ABB RAPID module: P43.mod

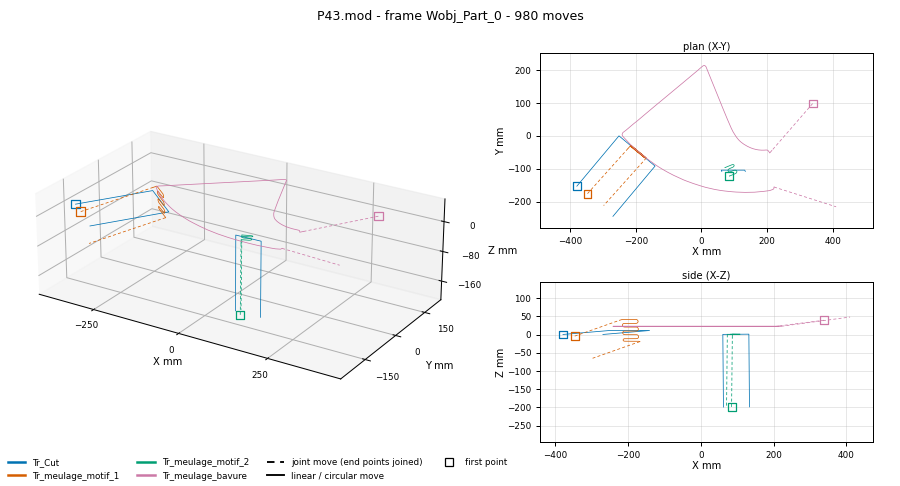
[picture p0: tool path of P43.mod in frame Wobj_Part_0, 980 of 990 moves have a stored position in this frame; points joined in program order, loops and branches not executed]
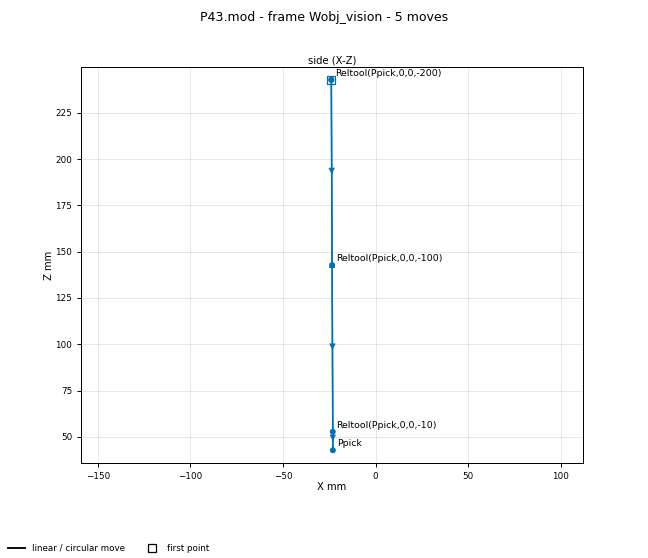
[picture p1: tool path of P43.mod in frame Wobj_vision, 5 of 990 moves have a stored position in this frame; points joined in program order, loops and branches not executed]
MODULE P43
	LOCAL CONST Speeddata vitesse_Tronconnage :=[10, 500, 0, 0];
	LOCAL CONST Robtarget Coupe_0 :=[[-192.24090625,-48.85296875,11.378640625],[0.632335428197394,0.648580331341073,0.281679878226159,0.316467859736843],[0,0,0,0],[8.999999E+09,8.999999E+09,8.999999E+09,8.999999E+09,8.999999E+09,8.999999E+09]];
	LOCAL CONST Robtarget Coupe_1 :=[[91.171640625,-104.02940625,0.997809143066406],[0.704150064324628,-0.0071021341686035,-0.709980726051425,0.00704380844178293],[0,0,0,0],[8.999999E+09,8.999999E+09,8.999999E+09,8.999999E+09,8.999999E+09,8.999999E+09]];
	LOCAL CONST Robtarget Tr_meulage_motif_1_App1 :=[[-346.886304833048,-175.614309992593,-4.01447746289841],[0.732123189175605,-0.57971865199821,0.222030212103854,-0.280400615744397],[0,0,0,0],[8.999999E+09,8.999999E+09,8.999999E+09,8.999999E+09,8.999999E+09,8.999999E+09]];
	LOCAL CONST Robtarget Tr_meulage_motif_1_App2 :=[[-223.345669929152,-37.9904471402547,39.5444929237301],[0.732123189175605,-0.57971865199821,0.222030212103854,-0.280400615744397],[0,0,0,0],[8.999999E+09,8.999999E+09,8.999999E+09,8.999999E+09,8.999999E+09,8.999999E+09]];
	LOCAL CONST Robtarget Tr_meulage_motif_1_P0 :=[[-216.84353125,-30.7470859375,41.8370703125],[0.732123189175605,-0.57971865199821,0.222030212103854,-0.280400615744397],[0,0,0,0],[8.999999E+09,8.999999E+09,8.999999E+09,8.999999E+09,8.999999E+09,8.999999E+09]];
	LOCAL CONST Robtarget Tr_meulage_motif_1_P1 :=[[-216.071953125,-31.38321875,41.837171875],[0.732123189175605,-0.57971865199821,0.222030212103854,-0.280400615744397],[0,0,0,0],[8.999999E+09,8.999999E+09,8.999999E+09,8.999999E+09,8.999999E+09,8.999999E+09]];
	LOCAL CONST Robtarget Tr_meulage_motif_1_P2 :=[[-215.300375,-32.0193515625,41.83726953125],[0.732123189175605,-0.57971865199821,0.222030212103854,-0.280400615744397],[0,0,0,0],[8.999999E+09,8.999999E+09,8.999999E+09,8.999999E+09,8.999999E+09,8.999999E+09]];
	LOCAL CONST Robtarget Tr_meulage_motif_1_P3 :=[[-214.52878125,-32.655486328125,41.8373671875],[0.732123189175605,-0.57971865199821,0.222030212103854,-0.280400615744397],[0,0,0,0],[8.999999E+09,8.999999E+09,8.999999E+09,8.999999E+09,8.999999E+09,8.999999E+09]];
	LOCAL CONST Robtarget Tr_meulage_motif_1_P4 :=[[-213.757203125,-33.2916171875,41.83746484375],[0.732123189175605,-0.57971865199821,0.222030212103854,-0.280400615744397],[0,0,0,0],[8.999999E+09,8.999999E+09,8.999999E+09,8.999999E+09,8.999999E+09,8.999999E+09]];
	LOCAL CONST Robtarget Tr_meulage_motif_1_P5 :=[[-212.985625,-33.92775390625,41.8375625],[0.732123189175605,-0.57971865199821,0.222030212103854,-0.280400615744397],[0,0,0,0],[8.999999E+09,8.999999E+09,8.999999E+09,8.999999E+09,8.999999E+09,8.999999E+09]];
	LOCAL CONST Robtarget Tr_meulage_motif_1_P6 :=[[-212.214046875,-34.56388671875,41.8376640625],[0.732123189175605,-0.57971865199821,0.222030212103854,-0.280400615744397],[0,0,0,0],[8.999999E+09,8.999999E+09,8.999999E+09,8.999999E+09,8.999999E+09,8.999999E+09]];
	LOCAL CONST Robtarget Tr_meulage_motif_1_P7 :=[[-211.44246875,-35.20001953125,41.83776171875],[0.732123189175605,-0.57971865199821,0.222030212103854,-0.280400615744397],[0,0,0,0],[8.999999E+09,8.999999E+09,8.999999E+09,8.999999E+09,8.999999E+09,8.999999E+09]];
	LOCAL CONST Robtarget Tr_meulage_motif_1_P8 :=[[-210.670890625,-35.83615234375,41.837859375],[0.732123189175605,-0.57971865199821,0.222030212103854,-0.280400615744397],[0,0,0,0],[8.999999E+09,8.999999E+09,8.999999E+09,8.999999E+09,8.999999E+09,8.999999E+09]];
	LOCAL CONST Robtarget Tr_meulage_motif_1_P9 :=[[-209.8993125,-36.47228515625,41.83795703125],[0.732123189175605,-0.57971865199821,0.222030212103854,-0.280400615744397],[0,0,0,0],[8.999999E+09,8.999999E+09,8.999999E+09,8.999999E+09,8.999999E+09,8.999999E+09]];
	LOCAL CONST Robtarget Tr_meulage_motif_1_P10 :=[[-209.127734375,-37.10841796875,41.8380546875],[0.732123189175605,-0.57971865199821,0.222030212103854,-0.280400615744397],[0,0,0,0],[8.999999E+09,8.999999E+09,8.999999E+09,8.999999E+09,8.999999E+09,8.999999E+09]];
	LOCAL CONST Robtarget Tr_meulage_motif_1_P11 :=[[-208.35615625,-37.74455078125,41.83815625],[0.732123189175605,-0.57971865199821,0.222030212103854,-0.280400615744397],[0,0,0,0],[8.999999E+09,8.999999E+09,8.999999E+09,8.999999E+09,8.999999E+09,8.999999E+09]];
	LOCAL CONST Robtarget Tr_meulage_motif_1_P12 :=[[-207.584578125,-38.38068359375,41.83825390625],[0.732123189175605,-0.57971865199821,0.222030212103854,-0.280400615744397],[0,0,0,0],[8.999999E+09,8.999999E+09,8.999999E+09,8.999999E+09,8.999999E+09,8.999999E+09]];
	LOCAL CONST Robtarget Tr_meulage_motif_1_P13 :=[[-206.813,-39.01681640625,41.8383515625],[0.732123189175605,-0.57971865199821,0.222030212103854,-0.280400615744397],[0,0,0,0],[8.999999E+09,8.999999E+09,8.999999E+09,8.999999E+09,8.999999E+09,8.999999E+09]];
	LOCAL CONST Robtarget Tr_meulage_motif_1_P14 :=[[-206.041421875,-39.65294921875,41.83844921875],[0.732123189175605,-0.57971865199821,0.222030212103854,-0.280400615744397],[0,0,0,0],[8.999999E+09,8.999999E+09,8.999999E+09,8.999999E+09,8.999999E+09,8.999999E+09]];
	LOCAL CONST Robtarget Tr_meulage_motif_1_P15 :=[[-205.26984375,-40.2890859375,41.83855078125],[0.732123189175605,-0.57971865199821,0.222030212103854,-0.280400615744397],[0,0,0,0],[8.999999E+09,8.999999E+09,8.999999E+09,8.999999E+09,8.999999E+09,8.999999E+09]];
	LOCAL CONST Robtarget Tr_meulage_motif_1_P16 :=[[-204.498265625,-40.92521875,41.8386484375],[0.732123189175605,-0.57971865199821,0.222030212103854,-0.280400615744397],[0,0,0,0],[8.999999E+09,8.999999E+09,8.999999E+09,8.999999E+09,8.999999E+09,8.999999E+09]];
	LOCAL CONST Robtarget Tr_meulage_motif_1_P17 :=[[-203.726671875,-41.5613515625,41.83874609375],[0.732123189175605,-0.57971865199821,0.222030212103854,-0.280400615744397],[0,0,0,0],[8.999999E+09,8.999999E+09,8.999999E+09,8.999999E+09,8.999999E+09,8.999999E+09]];
	LOCAL CONST Robtarget Tr_meulage_motif_1_P18 :=[[-202.95509375,-42.197484375,41.83884375],[0.732123189175605,-0.57971865199821,0.222030212103854,-0.280400615744397],[0,0,0,0],[8.999999E+09,8.999999E+09,8.999999E+09,8.999999E+09,8.999999E+09,8.999999E+09]];
	LOCAL CONST Robtarget Tr_meulage_motif_1_P19 :=[[-202.183515625,-42.8336171875,41.83894140625],[0.732123189175605,-0.57971865199821,0.222030212103854,-0.280400615744397],[0,0,0,0],[8.999999E+09,8.999999E+09,8.999999E+09,8.999999E+09,8.999999E+09,8.999999E+09]];
	LOCAL CONST Robtarget Tr_meulage_motif_1_P20 :=[[-201.4119375,-43.46975,41.83904296875],[0.732123189175605,-0.57971865199821,0.222030212103854,-0.280400615744397],[0,0,0,0],[8.999999E+09,8.999999E+09,8.999999E+09,8.999999E+09,8.999999E+09,8.999999E+09]];
	LOCAL CONST Robtarget Tr_meulage_motif_1_P21 :=[[-200.640359375,-44.1058828125,41.839140625],[0.732123189175605,-0.57971865199821,0.222030212103854,-0.280400615744397],[0,0,0,0],[8.999999E+09,8.999999E+09,8.999999E+09,8.999999E+09,8.999999E+09,8.999999E+09]];
	LOCAL CONST Robtarget Tr_meulage_motif_1_P22 :=[[-199.86878125,-44.742015625,41.83923828125],[0.732123189175605,-0.57971865199821,0.222030212103854,-0.280400615744397],[0,0,0,0],[8.999999E+09,8.999999E+09,8.999999E+09,8.999999E+09,8.999999E+09,8.999999E+09]];
	LOCAL CONST Robtarget Tr_meulage_motif_1_P23 :=[[-199.097203125,-45.3781484375,41.8393359375],[0.732123189175605,-0.57971865199821,0.222030212103854,-0.280400615744397],[0,0,0,0],[8.999999E+09,8.999999E+09,8.999999E+09,8.999999E+09,8.999999E+09,8.999999E+09]];
	LOCAL CONST Robtarget Tr_meulage_motif_1_P24 :=[[-198.325625,-46.01428515625,41.83943359375],[0.732123189175605,-0.57971865199821,0.222030212103854,-0.280400615744397],[0,0,0,0],[8.999999E+09,8.999999E+09,8.999999E+09,8.999999E+09,8.999999E+09,8.999999E+09]];
	LOCAL CONST Robtarget Tr_meulage_motif_1_P25 :=[[-197.554046875,-46.65041796875,41.83953515625],[0.732123189175605,-0.57971865199821,0.222030212103854,-0.280400615744397],[0,0,0,0],[8.999999E+09,8.999999E+09,8.999999E+09,8.999999E+09,8.999999E+09,8.999999E+09]];
	LOCAL CONST Robtarget Tr_meulage_motif_1_P26 :=[[-196.78246875,-47.28655078125,41.8396328125],[0.732123189175605,-0.57971865199821,0.222030212103854,-0.280400615744397],[0,0,0,0],[8.999999E+09,8.999999E+09,8.999999E+09,8.999999E+09,8.999999E+09,8.999999E+09]];
	LOCAL CONST Robtarget Tr_meulage_motif_1_P27 :=[[-196.010890625,-47.92268359375,41.83973046875],[0.732123189175605,-0.57971865199821,0.222030212103854,-0.280400615744397],[0,0,0,0],[8.999999E+09,8.999999E+09,8.999999E+09,8.999999E+09,8.999999E+09,8.999999E+09]];
	LOCAL CONST Robtarget Tr_meulage_motif_1_P28 :=[[-195.2393125,-48.55881640625,41.839828125],[0.732123189175605,-0.57971865199821,0.222030212103854,-0.280400615744397],[0,0,0,0],[8.999999E+09,8.999999E+09,8.999999E+09,8.999999E+09,8.999999E+09,8.999999E+09]];
	LOCAL CONST Robtarget Tr_meulage_motif_1_P29 :=[[-194.467734375,-49.19494921875,41.83992578125],[0.732123189175605,-0.57971865199821,0.222030212103854,-0.280400615744397],[0,0,0,0],[8.999999E+09,8.999999E+09,8.999999E+09,8.999999E+09,8.999999E+09,8.999999E+09]];
	LOCAL CONST Robtarget Tr_meulage_motif_1_P30 :=[[-193.69615625,-49.83108203125,41.84002734375],[0.732123189175605,-0.57971865199821,0.222030212103854,-0.280400615744397],[0,0,0,0],[8.999999E+09,8.999999E+09,8.999999E+09,8.999999E+09,8.999999E+09,8.999999E+09]];
	LOCAL CONST Robtarget Tr_meulage_motif_1_P31 :=[[-192.9245625,-50.46721484375,41.840125],[0.732123189175605,-0.57971865199821,0.222030212103854,-0.280400615744397],[0,0,0,0],[8.999999E+09,8.999999E+09,8.999999E+09,8.999999E+09,8.999999E+09,8.999999E+09]];
	LOCAL CONST Robtarget Tr_meulage_motif_1_P32 :=[[-192.152984375,-51.10334765625,41.84022265625],[0.732123189175605,-0.57971865199821,0.222030212103854,-0.280400615744397],[0,0,0,0],[8.999999E+09,8.999999E+09,8.999999E+09,8.999999E+09,8.999999E+09,8.999999E+09]];
	LOCAL CONST Robtarget Tr_meulage_motif_1_P33 :=[[-191.38140625,-51.73948046875,41.8403203125],[0.732123189175605,-0.57971865199821,0.222030212103854,-0.280400615744397],[0,0,0,0],[8.999999E+09,8.999999E+09,8.999999E+09,8.999999E+09,8.999999E+09,8.999999E+09]];
	LOCAL CONST Robtarget Tr_meulage_motif_1_P34 :=[[-190.609828125,-52.3756171875,41.840421875],[0.732123189175605,-0.57971865199821,0.222030212103854,-0.280400615744397],[0,0,0,0],[8.999999E+09,8.999999E+09,8.999999E+09,8.999999E+09,8.999999E+09,8.999999E+09]];
	LOCAL CONST Robtarget Tr_meulage_motif_1_P35 :=[[-189.83825,-53.01175,41.84051953125],[0.732123189175605,-0.57971865199821,0.222030212103854,-0.280400615744397],[0,0,0,0],[8.999999E+09,8.999999E+09,8.999999E+09,8.999999E+09,8.999999E+09,8.999999E+09]];
	LOCAL CONST Robtarget Tr_meulage_motif_1_P36 :=[[-189.066671875,-53.6478828125,41.8406171875],[0.732123189175605,-0.57971865199821,0.222030212103854,-0.280400615744397],[0,0,0,0],[8.999999E+09,8.999999E+09,8.999999E+09,8.999999E+09,8.999999E+09,8.999999E+09]];
	LOCAL CONST Robtarget Tr_meulage_motif_1_P37 :=[[-188.29509375,-54.284015625,41.84071484375],[0.732123189175605,-0.57971865199821,0.222030212103854,-0.280400615744397],[0,0,0,0],[8.999999E+09,8.999999E+09,8.999999E+09,8.999999E+09,8.999999E+09,8.999999E+09]];
	LOCAL CONST Robtarget Tr_meulage_motif_1_P38 :=[[-187.523515625,-54.9201484375,41.8408125],[0.732123189175605,-0.57971865199821,0.222030212103854,-0.280400615744397],[0,0,0,0],[8.999999E+09,8.999999E+09,8.999999E+09,8.999999E+09,8.999999E+09,8.999999E+09]];
	LOCAL CONST Robtarget Tr_meulage_motif_1_P39 :=[[-186.7519375,-55.55628125,41.8409140625],[0.732123189175605,-0.57971865199821,0.222030212103854,-0.280400615744397],[0,0,0,0],[8.999999E+09,8.999999E+09,8.999999E+09,8.999999E+09,8.999999E+09,8.999999E+09]];
	LOCAL CONST Robtarget Tr_meulage_motif_1_P40 :=[[-185.980359375,-56.1924140625,41.84101171875],[0.732123189175605,-0.57971865199821,0.222030212103854,-0.280400615744397],[0,0,0,0],[8.999999E+09,8.999999E+09,8.999999E+09,8.999999E+09,8.999999E+09,8.999999E+09]];
	LOCAL CONST Robtarget Tr_meulage_motif_1_P41 :=[[-185.20878125,-56.828546875,41.841109375],[0.732123189175605,-0.57971865199821,0.222030212103854,-0.280400615744397],[0,0,0,0],[8.999999E+09,8.999999E+09,8.999999E+09,8.999999E+09,8.999999E+09,8.999999E+09]];
	LOCAL CONST Robtarget Tr_meulage_motif_1_P42 :=[[-184.437203125,-57.4646796875,41.84120703125],[0.732123189175605,-0.57971865199821,0.222030212103854,-0.280400615744397],[0,0,0,0],[8.999999E+09,8.999999E+09,8.999999E+09,8.999999E+09,8.999999E+09,8.999999E+09]];
	LOCAL CONST Robtarget Tr_meulage_motif_1_P43 :=[[-183.665625,-58.10081640625,41.8413046875],[0.732123189175605,-0.57971865199821,0.222030212103854,-0.280400615744397],[0,0,0,0],[8.999999E+09,8.999999E+09,8.999999E+09,8.999999E+09,8.999999E+09,8.999999E+09]];
	LOCAL CONST Robtarget Tr_meulage_motif_1_P44 :=[[-182.894046875,-58.73694921875,41.84140625],[0.732123189175605,-0.57971865199821,0.222030212103854,-0.280400615744397],[0,0,0,0],[8.999999E+09,8.999999E+09,8.999999E+09,8.999999E+09,8.999999E+09,8.999999E+09]];
	LOCAL CONST Robtarget Tr_meulage_motif_1_P45 :=[[-182.122453125,-59.37308203125,41.84150390625],[0.732123189175605,-0.57971865199821,0.222030212103854,-0.280400615744397],[0,0,0,0],[8.999999E+09,8.999999E+09,8.999999E+09,8.999999E+09,8.999999E+09,8.999999E+09]];
	LOCAL CONST Robtarget Tr_meulage_motif_1_P46 :=[[-181.350875,-60.00921484375,41.8416015625],[0.732123189175605,-0.57971865199821,0.222030212103854,-0.280400615744397],[0,0,0,0],[8.999999E+09,8.999999E+09,8.999999E+09,8.999999E+09,8.999999E+09,8.999999E+09]];
	LOCAL CONST Robtarget Tr_meulage_motif_1_P47 :=[[-180.579296875,-60.64534765625,41.84169921875],[0.732123189175605,-0.57971865199821,0.222030212103854,-0.280400615744397],[0,0,0,0],[8.999999E+09,8.999999E+09,8.999999E+09,8.999999E+09,8.999999E+09,8.999999E+09]];
	LOCAL CONST Robtarget Tr_meulage_motif_1_P48 :=[[-179.80771875,-61.28148046875,41.841796875],[0.732123189175605,-0.57971865199821,0.222030212103854,-0.280400615744397],[0,0,0,0],[8.999999E+09,8.999999E+09,8.999999E+09,8.999999E+09,8.999999E+09,8.999999E+09]];
	LOCAL CONST Robtarget Tr_meulage_motif_1_P49 :=[[-179.036140625,-61.91761328125,41.8418984375],[0.732123189175605,-0.57971865199821,0.222030212103854,-0.280400615744397],[0,0,0,0],[8.999999E+09,8.999999E+09,8.999999E+09,8.999999E+09,8.999999E+09,8.999999E+09]];
	LOCAL CONST Robtarget Tr_meulage_motif_1_P50 :=[[-178.2645625,-62.55374609375,41.84199609375],[0.732123189175605,-0.57971865199821,0.222030212103854,-0.280400615744397],[0,0,0,0],[8.999999E+09,8.999999E+09,8.999999E+09,8.999999E+09,8.999999E+09,8.999999E+09]];
	LOCAL CONST Robtarget Tr_meulage_motif_1_P51 :=[[-177.49484375,-63.18045703125,41.73166796875],[0.732123189175605,-0.57971865199821,0.222030212103854,-0.280400615744397],[0,0,0,0],[8.999999E+09,8.999999E+09,8.999999E+09,8.999999E+09,8.999999E+09,8.999999E+09]];
	LOCAL CONST Robtarget Tr_meulage_motif_1_P52 :=[[-176.757125,-63.77359375,41.52089453125],[0.732123189175605,-0.57971865199821,0.222030212103854,-0.280400615744397],[0,0,0,0],[8.999999E+09,8.999999E+09,8.999999E+09,8.999999E+09,8.999999E+09,8.999999E+09]];
	LOCAL CONST Robtarget Tr_meulage_motif_1_P53 :=[[-176.089640625,-64.3045,41.249546875],[0.732123189175605,-0.57971865199821,0.222030212103854,-0.280400615744397],[0,0,0,0],[8.999999E+09,8.999999E+09,8.999999E+09,8.999999E+09,8.999999E+09,8.999999E+09]];
	LOCAL CONST Robtarget Tr_meulage_motif_1_P54 :=[[-175.5013125,-64.7698515625,40.9741015625],[0.732123189175605,-0.57971865199821,0.222030212103854,-0.280400615744397],[0,0,0,0],[8.999999E+09,8.999999E+09,8.999999E+09,8.999999E+09,8.999999E+09,8.999999E+09]];
	LOCAL CONST Robtarget Tr_meulage_motif_1_P55 :=[[-174.630125,-65.444125,40.35901953125],[0.732123189175605,-0.57971865199821,0.222030212103854,-0.280400615744397],[0,0,0,0],[8.999999E+09,8.999999E+09,8.999999E+09,8.999999E+09,8.999999E+09,8.999999E+09]];
	LOCAL CONST Robtarget Tr_meulage_motif_1_P56 :=[[-173.810359375,-66.0594765625,39.51275390625],[0.732123189175605,-0.57971865199821,0.222030212103854,-0.280400615744397],[0,0,0,0],[8.999999E+09,8.999999E+09,8.999999E+09,8.999999E+09,8.999999E+09,8.999999E+09]];
	LOCAL CONST Robtarget Tr_meulage_motif_1_P57 :=[[-173.120359375,-66.5552421875,38.490515625],[0.732123189175605,-0.57971865199821,0.222030212103854,-0.280400615744397],[0,0,0,0],[8.999999E+09,8.999999E+09,8.999999E+09,8.999999E+09,8.999999E+09,8.999999E+09]];
	LOCAL CONST Robtarget Tr_meulage_motif_1_P58 :=[[-172.704515625,-66.8184140625,37.3760703125],[0.732123189175605,-0.57971865199821,0.222030212103854,-0.280400615744397],[0,0,0,0],[8.999999E+09,8.999999E+09,8.999999E+09,8.999999E+09,8.999999E+09,8.999999E+09]];
	LOCAL CONST Robtarget Tr_meulage_motif_1_P59 :=[[-172.659203125,-66.80609375,36.68116015625],[0.732123189175605,-0.57971865199821,0.222030212103854,-0.280400615744397],[0,0,0,0],[8.999999E+09,8.999999E+09,8.999999E+09,8.999999E+09,8.999999E+09,8.999999E+09]];
	LOCAL CONST Robtarget Tr_meulage_motif_1_P60 :=[[-172.635984375,-66.77803125,36.0209140625],[0.732123189175605,-0.57971865199821,0.222030212103854,-0.280400615744397],[0,0,0,0],[8.999999E+09,8.999999E+09,8.999999E+09,8.999999E+09,8.999999E+09,8.999999E+09]];
	LOCAL CONST Robtarget Tr_meulage_motif_1_P61 :=[[-172.655109375,-66.7150625,35.3608203125],[0.732123189175605,-0.57971865199821,0.222030212103854,-0.280400615744397],[0,0,0,0],[8.999999E+09,8.999999E+09,8.999999E+09,8.999999E+09,8.999999E+09,8.999999E+09]];
	LOCAL CONST Robtarget Tr_meulage_motif_1_P62 :=[[-173.000828125,-66.351375,34.26069140625],[0.732123189175605,-0.57971865199821,0.222030212103854,-0.280400615744397],[0,0,0,0],[8.999999E+09,8.999999E+09,8.999999E+09,8.999999E+09,8.999999E+09,8.999999E+09]];
	LOCAL CONST Robtarget Tr_meulage_motif_1_P63 :=[[-173.6264375,-65.763734375,33.25551171875],[0.732123189175605,-0.57971865199821,0.222030212103854,-0.280400615744397],[0,0,0,0],[8.999999E+09,8.999999E+09,8.999999E+09,8.999999E+09,8.999999E+09,8.999999E+09]];
	LOCAL CONST Robtarget Tr_meulage_motif_1_P64 :=[[-174.38696875,-65.07753125,32.427794921875],[0.732123189175605,-0.57971865199821,0.222030212103854,-0.280400615744397],[0,0,0,0],[8.999999E+09,8.999999E+09,8.999999E+09,8.999999E+09,8.999999E+09,8.999999E+09]];
	LOCAL CONST Robtarget Tr_meulage_motif_1_P65 :=[[-174.90321875,-64.62365625,32.032578125],[0.732123189175605,-0.57971865199821,0.222030212103854,-0.280400615744397],[0,0,0,0],[8.999999E+09,8.999999E+09,8.999999E+09,8.999999E+09,8.999999E+09,8.999999E+09]];
	LOCAL CONST Robtarget Tr_meulage_motif_1_P66 :=[[-175.77971875,-63.86622265625,31.545671875],[0.732123189175605,-0.57971865199821,0.222030212103854,-0.280400615744397],[0,0,0,0],[8.999999E+09,8.999999E+09,8.999999E+09,8.999999E+09,8.999999E+09,8.999999E+09]];
	LOCAL CONST Robtarget Tr_meulage_motif_1_P67 :=[[-176.422453125,-63.31746484375,31.281896484375],[0.732123189175605,-0.57971865199821,0.222030212103854,-0.280400615744397],[0,0,0,0],[8.999999E+09,8.999999E+09,8.999999E+09,8.999999E+09,8.999999E+09,8.999999E+09]];
	LOCAL CONST Robtarget Tr_meulage_motif_1_P68 :=[[-177.134375,-62.71591015625,31.077646484375],[0.732123189175605,-0.57971865199821,0.222030212103854,-0.280400615744397],[0,0,0,0],[8.999999E+09,8.999999E+09,8.999999E+09,8.999999E+09,8.999999E+09,8.999999E+09]];
	LOCAL CONST Robtarget Tr_meulage_motif_1_P69 :=[[-177.887921875,-62.0868984375,30.96912109375],[0.732123189175605,-0.57971865199821,0.222030212103854,-0.280400615744397],[0,0,0,0],[8.999999E+09,8.999999E+09,8.999999E+09,8.999999E+09,8.999999E+09,8.999999E+09]];
	LOCAL CONST Robtarget Tr_meulage_motif_1_P70 :=[[-178.649875,-61.45080078125,30.85859765625],[0.732123189175605,-0.57971865199821,0.222030212103854,-0.280400615744397],[0,0,0,0],[8.999999E+09,8.999999E+09,8.999999E+09,8.999999E+09,8.999999E+09,8.999999E+09]];
	LOCAL CONST Robtarget Tr_meulage_motif_1_P71 :=[[-179.421453125,-60.81466796875,30.858498046875],[0.732123189175605,-0.57971865199821,0.222030212103854,-0.280400615744397],[0,0,0,0],[8.999999E+09,8.999999E+09,8.999999E+09,8.999999E+09,8.999999E+09,8.999999E+09]];
	LOCAL CONST Robtarget Tr_meulage_motif_1_P72 :=[[-180.19303125,-60.17853515625,30.858400390625],[0.732123189175605,-0.57971865199821,0.222030212103854,-0.280400615744397],[0,0,0,0],[8.999999E+09,8.999999E+09,8.999999E+09,8.999999E+09,8.999999E+09,8.999999E+09]];
	LOCAL CONST Robtarget Tr_meulage_motif_1_P73 :=[[-180.964609375,-59.54240234375,30.85830078125],[0.732123189175605,-0.57971865199821,0.222030212103854,-0.280400615744397],[0,0,0,0],[8.999999E+09,8.999999E+09,8.999999E+09,8.999999E+09,8.999999E+09,8.999999E+09]];
	LOCAL CONST Robtarget Tr_meulage_motif_1_P74 :=[[-181.7361875,-58.90626953125,30.858203125],[0.732123189175605,-0.57971865199821,0.222030212103854,-0.280400615744397],[0,0,0,0],[8.999999E+09,8.999999E+09,8.999999E+09,8.999999E+09,8.999999E+09,8.999999E+09]];
	LOCAL CONST Robtarget Tr_meulage_motif_1_P75 :=[[-182.507765625,-58.27013671875,30.858103515625],[0.732123189175605,-0.57971865199821,0.222030212103854,-0.280400615744397],[0,0,0,0],[8.999999E+09,8.999999E+09,8.999999E+09,8.999999E+09,8.999999E+09,8.999999E+09]];
	LOCAL CONST Robtarget Tr_meulage_motif_1_P76 :=[[-183.279359375,-57.63400390625,30.858005859375],[0.732123189175605,-0.57971865199821,0.222030212103854,-0.280400615744397],[0,0,0,0],[8.999999E+09,8.999999E+09,8.999999E+09,8.999999E+09,8.999999E+09,8.999999E+09]];
	LOCAL CONST Robtarget Tr_meulage_motif_1_P77 :=[[-184.0509375,-56.99787109375,30.857908203125],[0.732123189175605,-0.57971865199821,0.222030212103854,-0.280400615744397],[0,0,0,0],[8.999999E+09,8.999999E+09,8.999999E+09,8.999999E+09,8.999999E+09,8.999999E+09]];
	LOCAL CONST Robtarget Tr_meulage_motif_1_P78 :=[[-184.822515625,-56.36173828125,30.85780859375],[0.732123189175605,-0.57971865199821,0.222030212103854,-0.280400615744397],[0,0,0,0],[8.999999E+09,8.999999E+09,8.999999E+09,8.999999E+09,8.999999E+09,8.999999E+09]];
	LOCAL CONST Robtarget Tr_meulage_motif_1_P79 :=[[-185.59409375,-55.7256015625,30.8577109375],[0.732123189175605,-0.57971865199821,0.222030212103854,-0.280400615744397],[0,0,0,0],[8.999999E+09,8.999999E+09,8.999999E+09,8.999999E+09,8.999999E+09,8.999999E+09]];
	LOCAL CONST Robtarget Tr_meulage_motif_1_P80 :=[[-186.365671875,-55.08946875,30.857611328125],[0.732123189175605,-0.57971865199821,0.222030212103854,-0.280400615744397],[0,0,0,0],[8.999999E+09,8.999999E+09,8.999999E+09,8.999999E+09,8.999999E+09,8.999999E+09]];
	LOCAL CONST Robtarget Tr_meulage_motif_1_P81 :=[[-187.13725,-54.4533359375,30.857513671875],[0.732123189175605,-0.57971865199821,0.222030212103854,-0.280400615744397],[0,0,0,0],[8.999999E+09,8.999999E+09,8.999999E+09,8.999999E+09,8.999999E+09,8.999999E+09]];
	LOCAL CONST Robtarget Tr_meulage_motif_1_P82 :=[[-187.908828125,-53.817203125,30.857416015625],[0.732123189175605,-0.57971865199821,0.222030212103854,-0.280400615744397],[0,0,0,0],[8.999999E+09,8.999999E+09,8.999999E+09,8.999999E+09,8.999999E+09,8.999999E+09]];
	LOCAL CONST Robtarget Tr_meulage_motif_1_P83 :=[[-188.68040625,-53.1810703125,30.85731640625],[0.732123189175605,-0.57971865199821,0.222030212103854,-0.280400615744397],[0,0,0,0],[8.999999E+09,8.999999E+09,8.999999E+09,8.999999E+09,8.999999E+09,8.999999E+09]];
	LOCAL CONST Robtarget Tr_meulage_motif_1_P84 :=[[-189.451984375,-52.5449375,30.85721875],[0.732123189175605,-0.57971865199821,0.222030212103854,-0.280400615744397],[0,0,0,0],[8.999999E+09,8.999999E+09,8.999999E+09,8.999999E+09,8.999999E+09,8.999999E+09]];
	LOCAL CONST Robtarget Tr_meulage_motif_1_P85 :=[[-190.2235625,-51.9088046875,30.857119140625],[0.732123189175605,-0.57971865199821,0.222030212103854,-0.280400615744397],[0,0,0,0],[8.999999E+09,8.999999E+09,8.999999E+09,8.999999E+09,8.999999E+09,8.999999E+09]];
	LOCAL CONST Robtarget Tr_meulage_motif_1_P86 :=[[-190.995140625,-51.272671875,30.857021484375],[0.732123189175605,-0.57971865199821,0.222030212103854,-0.280400615744397],[0,0,0,0],[8.999999E+09,8.999999E+09,8.999999E+09,8.999999E+09,8.999999E+09,8.999999E+09]];
	LOCAL CONST Robtarget Tr_meulage_motif_1_P87 :=[[-191.76671875,-50.6365390625,30.856921875],[0.732123189175605,-0.57971865199821,0.222030212103854,-0.280400615744397],[0,0,0,0],[8.999999E+09,8.999999E+09,8.999999E+09,8.999999E+09,8.999999E+09,8.999999E+09]];
	LOCAL CONST Robtarget Tr_meulage_motif_1_P88 :=[[-192.538296875,-50.00040625,30.85682421875],[0.732123189175605,-0.57971865199821,0.222030212103854,-0.280400615744397],[0,0,0,0],[8.999999E+09,8.999999E+09,8.999999E+09,8.999999E+09,8.999999E+09,8.999999E+09]];
	LOCAL CONST Robtarget Tr_meulage_motif_1_P89 :=[[-193.309875,-49.36426953125,30.8567265625],[0.732123189175605,-0.57971865199821,0.222030212103854,-0.280400615744397],[0,0,0,0],[8.999999E+09,8.999999E+09,8.999999E+09,8.999999E+09,8.999999E+09,8.999999E+09]];
	LOCAL CONST Robtarget Tr_meulage_motif_1_P90 :=[[-194.08146875,-48.72813671875,30.856626953125],[0.732123189175605,-0.57971865199821,0.222030212103854,-0.280400615744397],[0,0,0,0],[8.999999E+09,8.999999E+09,8.999999E+09,8.999999E+09,8.999999E+09,8.999999E+09]];
	LOCAL CONST Robtarget Tr_meulage_motif_1_P91 :=[[-194.853046875,-48.09200390625,30.856529296875],[0.732123189175605,-0.57971865199821,0.222030212103854,-0.280400615744397],[0,0,0,0],[8.999999E+09,8.999999E+09,8.999999E+09,8.999999E+09,8.999999E+09,8.999999E+09]];
	LOCAL CONST Robtarget Tr_meulage_motif_1_P92 :=[[-195.624625,-47.45587109375,30.8564296875],[0.732123189175605,-0.57971865199821,0.222030212103854,-0.280400615744397],[0,0,0,0],[8.999999E+09,8.999999E+09,8.999999E+09,8.999999E+09,8.999999E+09,8.999999E+09]];
	LOCAL CONST Robtarget Tr_meulage_motif_1_P93 :=[[-196.396203125,-46.81973828125,30.85633203125],[0.732123189175605,-0.57971865199821,0.222030212103854,-0.280400615744397],[0,0,0,0],[8.999999E+09,8.999999E+09,8.999999E+09,8.999999E+09,8.999999E+09,8.999999E+09]];
	LOCAL CONST Robtarget Tr_meulage_motif_1_P94 :=[[-197.16778125,-46.18360546875,30.856234375],[0.732123189175605,-0.57971865199821,0.222030212103854,-0.280400615744397],[0,0,0,0],[8.999999E+09,8.999999E+09,8.999999E+09,8.999999E+09,8.999999E+09,8.999999E+09]];
	LOCAL CONST Robtarget Tr_meulage_motif_1_P95 :=[[-197.939359375,-45.54747265625,30.856134765625],[0.732123189175605,-0.57971865199821,0.222030212103854,-0.280400615744397],[0,0,0,0],[8.999999E+09,8.999999E+09,8.999999E+09,8.999999E+09,8.999999E+09,8.999999E+09]];
	LOCAL CONST Robtarget Tr_meulage_motif_1_P96 :=[[-198.7109375,-44.91133984375,30.856037109375],[0.732123189175605,-0.57971865199821,0.222030212103854,-0.280400615744397],[0,0,0,0],[8.999999E+09,8.999999E+09,8.999999E+09,8.999999E+09,8.999999E+09,8.999999E+09]];
	LOCAL CONST Robtarget Tr_meulage_motif_1_P97 :=[[-199.482515625,-44.27520703125,30.8559375],[0.732123189175605,-0.57971865199821,0.222030212103854,-0.280400615744397],[0,0,0,0],[8.999999E+09,8.999999E+09,8.999999E+09,8.999999E+09,8.999999E+09,8.999999E+09]];
	LOCAL CONST Robtarget Tr_meulage_motif_1_P98 :=[[-200.25409375,-43.6390703125,30.85583984375],[0.732123189175605,-0.57971865199821,0.222030212103854,-0.280400615744397],[0,0,0,0],[8.999999E+09,8.999999E+09,8.999999E+09,8.999999E+09,8.999999E+09,8.999999E+09]];
	LOCAL CONST Robtarget Tr_meulage_motif_1_P99 :=[[-201.025671875,-43.0029375,30.855740234375],[0.732123189175605,-0.57971865199821,0.222030212103854,-0.280400615744397],[0,0,0,0],[8.999999E+09,8.999999E+09,8.999999E+09,8.999999E+09,8.999999E+09,8.999999E+09]];
	LOCAL CONST Robtarget Tr_meulage_motif_1_P100 :=[[-201.79725,-42.3668046875,30.855642578125],[0.732123189175605,-0.57971865199821,0.222030212103854,-0.280400615744397],[0,0,0,0],[8.999999E+09,8.999999E+09,8.999999E+09,8.999999E+09,8.999999E+09,8.999999E+09]];
	LOCAL CONST Robtarget Tr_meulage_motif_1_P101 :=[[-202.568828125,-41.730671875,30.855544921875],[0.732123189175605,-0.57971865199821,0.222030212103854,-0.280400615744397],[0,0,0,0],[8.999999E+09,8.999999E+09,8.999999E+09,8.999999E+09,8.999999E+09,8.999999E+09]];
	LOCAL CONST Robtarget Tr_meulage_motif_1_P102 :=[[-203.34040625,-41.0945390625,30.8554453125],[0.732123189175605,-0.57971865199821,0.222030212103854,-0.280400615744397],[0,0,0,0],[8.999999E+09,8.999999E+09,8.999999E+09,8.999999E+09,8.999999E+09,8.999999E+09]];
	LOCAL CONST Robtarget Tr_meulage_motif_1_P103 :=[[-204.111984375,-40.45840625,30.85534765625],[0.732123189175605,-0.57971865199821,0.222030212103854,-0.280400615744397],[0,0,0,0],[8.999999E+09,8.999999E+09,8.999999E+09,8.999999E+09,8.999999E+09,8.999999E+09]];
	LOCAL CONST Robtarget Tr_meulage_motif_1_P104 :=[[-204.883578125,-39.8222734375,30.855248046875],[0.732123189175605,-0.57971865199821,0.222030212103854,-0.280400615744397],[0,0,0,0],[8.999999E+09,8.999999E+09,8.999999E+09,8.999999E+09,8.999999E+09,8.999999E+09]];
	LOCAL CONST Robtarget Tr_meulage_motif_1_P105 :=[[-205.65515625,-39.186140625,30.855150390625],[0.732123189175605,-0.57971865199821,0.222030212103854,-0.280400615744397],[0,0,0,0],[8.999999E+09,8.999999E+09,8.999999E+09,8.999999E+09,8.999999E+09,8.999999E+09]];
	LOCAL CONST Robtarget Tr_meulage_motif_1_P106 :=[[-206.426734375,-38.5500078125,30.85505078125],[0.732123189175605,-0.57971865199821,0.222030212103854,-0.280400615744397],[0,0,0,0],[8.999999E+09,8.999999E+09,8.999999E+09,8.999999E+09,8.999999E+09,8.999999E+09]];
	LOCAL CONST Robtarget Tr_meulage_motif_1_P107 :=[[-207.1983125,-37.913875,30.854953125],[0.732123189175605,-0.57971865199821,0.222030212103854,-0.280400615744397],[0,0,0,0],[8.999999E+09,8.999999E+09,8.999999E+09,8.999999E+09,8.999999E+09,8.999999E+09]];
	LOCAL CONST Robtarget Tr_meulage_motif_1_P108 :=[[-207.969890625,-37.27773828125,30.85485546875],[0.732123189175605,-0.57971865199821,0.222030212103854,-0.280400615744397],[0,0,0,0],[8.999999E+09,8.999999E+09,8.999999E+09,8.999999E+09,8.999999E+09,8.999999E+09]];
	LOCAL CONST Robtarget Tr_meulage_motif_1_P109 :=[[-208.74146875,-36.64160546875,30.854755859375],[0.732123189175605,-0.57971865199821,0.222030212103854,-0.280400615744397],[0,0,0,0],[8.999999E+09,8.999999E+09,8.999999E+09,8.999999E+09,8.999999E+09,8.999999E+09]];
	LOCAL CONST Robtarget Tr_meulage_motif_1_P110 :=[[-209.513046875,-36.00547265625,30.854658203125],[0.732123189175605,-0.57971865199821,0.222030212103854,-0.280400615744397],[0,0,0,0],[8.999999E+09,8.999999E+09,8.999999E+09,8.999999E+09,8.999999E+09,8.999999E+09]];
	LOCAL CONST Robtarget Tr_meulage_motif_1_P111 :=[[-210.284625,-35.36933984375,30.85455859375],[0.732123189175605,-0.57971865199821,0.222030212103854,-0.280400615744397],[0,0,0,0],[8.999999E+09,8.999999E+09,8.999999E+09,8.999999E+09,8.999999E+09,8.999999E+09]];
	LOCAL CONST Robtarget Tr_meulage_motif_1_P112 :=[[-211.056203125,-34.73320703125,30.8544609375],[0.732123189175605,-0.57971865199821,0.222030212103854,-0.280400615744397],[0,0,0,0],[8.999999E+09,8.999999E+09,8.999999E+09,8.999999E+09,8.999999E+09,8.999999E+09]];
	LOCAL CONST Robtarget Tr_meulage_motif_1_P113 :=[[-211.81815625,-34.09711328125,30.7439375],[0.732123189175605,-0.57971865199821,0.222030212103854,-0.280400615744397],[0,0,0,0],[8.999999E+09,8.999999E+09,8.999999E+09,8.999999E+09,8.999999E+09,8.999999E+09]];
	LOCAL CONST Robtarget Tr_meulage_motif_1_P114 :=[[-212.541046875,-33.48605078125,30.5329765625],[0.732123189175605,-0.57971865199821,0.222030212103854,-0.280400615744397],[0,0,0,0],[8.999999E+09,8.999999E+09,8.999999E+09,8.999999E+09,8.999999E+09,8.999999E+09]];
	LOCAL CONST Robtarget Tr_meulage_motif_1_P115 :=[[-213.1894375,-32.9320703125,30.261462890625],[0.732123189175605,-0.57971865199821,0.222030212103854,-0.280400615744397],[0,0,0,0],[8.999999E+09,8.999999E+09,8.999999E+09,8.999999E+09,8.999999E+09,8.999999E+09]];
	LOCAL CONST Robtarget Tr_meulage_motif_1_P116 :=[[-213.727734375,-32.4665546875,29.957697265625],[0.732123189175605,-0.57971865199821,0.222030212103854,-0.280400615744397],[0,0,0,0],[8.999999E+09,8.999999E+09,8.999999E+09,8.999999E+09,8.999999E+09,8.999999E+09]];
	LOCAL CONST Robtarget Tr_meulage_motif_1_P117 :=[[-214.502640625,-31.78037890625,29.2960703125],[0.732123189175605,-0.57971865199821,0.222030212103854,-0.280400615744397],[0,0,0,0],[8.999999E+09,8.999999E+09,8.999999E+09,8.999999E+09,8.999999E+09,8.999999E+09]];
	LOCAL CONST Robtarget Tr_meulage_motif_1_P118 :=[[-215.166890625,-31.168349609375,28.3954140625],[0.732123189175605,-0.57971865199821,0.222030212103854,-0.280400615744397],[0,0,0,0],[8.999999E+09,8.999999E+09,8.999999E+09,8.999999E+09,8.999999E+09,8.999999E+09]];
	LOCAL CONST Robtarget Tr_meulage_motif_1_P119 :=[[-215.5429375,-30.783646484375,27.35091796875],[0.732123189175605,-0.57971865199821,0.222030212103854,-0.280400615744397],[0,0,0,0],[8.999999E+09,8.999999E+09,8.999999E+09,8.999999E+09,8.999999E+09,8.999999E+09]];
	LOCAL CONST Robtarget Tr_meulage_motif_1_P120 :=[[-215.66115625,-30.63668359375,26.658732421875],[0.732123189175605,-0.57971865199821,0.222030212103854,-0.280400615744397],[0,0,0,0],[8.999999E+09,8.999999E+09,8.999999E+09,8.999999E+09,8.999999E+09,8.999999E+09]];
	LOCAL CONST Robtarget Tr_meulage_motif_1_P121 :=[[-215.683390625,-30.56339453125,25.889896484375],[0.732123189175605,-0.57971865199821,0.222030212103854,-0.280400615744397],[0,0,0,0],[8.999999E+09,8.999999E+09,8.999999E+09,8.999999E+09,8.999999E+09,8.999999E+09]];
	LOCAL CONST Robtarget Tr_meulage_motif_1_P122 :=[[-215.604703125,-30.573302734375,25.1211953125],[0.732123189175605,-0.57971865199821,0.222030212103854,-0.280400615744397],[0,0,0,0],[8.999999E+09,8.999999E+09,8.999999E+09,8.999999E+09,8.999999E+09,8.999999E+09]];
	LOCAL CONST Robtarget Tr_meulage_motif_1_P123 :=[[-215.24203125,-30.793189453125,24.014669921875],[0.732123189175605,-0.57971865199821,0.222030212103854,-0.280400615744397],[0,0,0,0],[8.999999E+09,8.999999E+09,8.999999E+09,8.999999E+09,8.999999E+09,8.999999E+09]];
	LOCAL CONST Robtarget Tr_meulage_motif_1_P124 :=[[-214.901796875,-31.031892578125,23.429912109375],[0.732123189175605,-0.57971865199821,0.222030212103854,-0.280400615744397],[0,0,0,0],[8.999999E+09,8.999999E+09,8.999999E+09,8.999999E+09,8.999999E+09,8.999999E+09]];
	LOCAL CONST Robtarget Tr_meulage_motif_1_P125 :=[[-214.18615625,-31.55857421875,22.544220703125],[0.732123189175605,-0.57971865199821,0.222030212103854,-0.280400615744397],[0,0,0,0],[8.999999E+09,8.999999E+09,8.999999E+09,8.999999E+09,8.999999E+09,8.999999E+09]];
	LOCAL CONST Robtarget Tr_meulage_motif_1_P126 :=[[-213.719703125,-31.913568359375,22.130595703125],[0.732123189175605,-0.57971865199821,0.222030212103854,-0.280400615744397],[0,0,0,0],[8.999999E+09,8.999999E+09,8.999999E+09,8.999999E+09,8.999999E+09,8.999999E+09]];
	LOCAL CONST Robtarget Tr_meulage_motif_1_P127 :=[[-212.838046875,-32.601615234375,21.5874375],[0.732123189175605,-0.57971865199821,0.222030212103854,-0.280400615744397],[0,0,0,0],[8.999999E+09,8.999999E+09,8.999999E+09,8.999999E+09,8.999999E+09,8.999999E+09]];
	LOCAL CONST Robtarget Tr_meulage_motif_1_P128 :=[[-212.19065625,-33.11426171875,21.29246875],[0.732123189175605,-0.57971865199821,0.222030212103854,-0.280400615744397],[0,0,0,0],[8.999999E+09,8.999999E+09,8.999999E+09,8.999999E+09,8.999999E+09,8.999999E+09]];
	LOCAL CONST Robtarget Tr_meulage_motif_1_P129 :=[[-211.464359375,-33.6984609375,21.088400390625],[0.732123189175605,-0.57971865199821,0.222030212103854,-0.280400615744397],[0,0,0,0],[8.999999E+09,8.999999E+09,8.999999E+09,8.999999E+09,8.999999E+09,8.999999E+09]];
	LOCAL CONST Robtarget Tr_meulage_motif_1_P130 :=[[-210.703203125,-34.3182578125,20.980068359375],[0.732123189175605,-0.57971865199821,0.222030212103854,-0.280400615744397],[0,0,0,0],[8.999999E+09,8.999999E+09,8.999999E+09,8.999999E+09,8.999999E+09,8.999999E+09]];
	LOCAL CONST Robtarget Tr_meulage_motif_1_P131 :=[[-209.93346875,-34.94496484375,20.869740234375],[0.732123189175605,-0.57971865199821,0.222030212103854,-0.280400615744397],[0,0,0,0],[8.999999E+09,8.999999E+09,8.999999E+09,8.999999E+09,8.999999E+09,8.999999E+09]];
	LOCAL CONST Robtarget Tr_meulage_motif_1_P132 :=[[-209.161890625,-35.58109765625,20.86983984375],[0.732123189175605,-0.57971865199821,0.222030212103854,-0.280400615744397],[0,0,0,0],[8.999999E+09,8.999999E+09,8.999999E+09,8.999999E+09,8.999999E+09,8.999999E+09]];
	LOCAL CONST Robtarget Tr_meulage_motif_1_P133 :=[[-208.3903125,-36.217234375,20.8699375],[0.732123189175605,-0.57971865199821,0.222030212103854,-0.280400615744397],[0,0,0,0],[8.999999E+09,8.999999E+09,8.999999E+09,8.999999E+09,8.999999E+09,8.999999E+09]];
	LOCAL CONST Robtarget Tr_meulage_motif_1_P134 :=[[-207.618734375,-36.8533671875,20.870037109375],[0.732123189175605,-0.57971865199821,0.222030212103854,-0.280400615744397],[0,0,0,0],[8.999999E+09,8.999999E+09,8.999999E+09,8.999999E+09,8.999999E+09,8.999999E+09]];
	LOCAL CONST Robtarget Tr_meulage_motif_1_P135 :=[[-206.84715625,-37.4895,20.870134765625],[0.732123189175605,-0.57971865199821,0.222030212103854,-0.280400615744397],[0,0,0,0],[8.999999E+09,8.999999E+09,8.999999E+09,8.999999E+09,8.999999E+09,8.999999E+09]];
	LOCAL CONST Robtarget Tr_meulage_motif_1_P136 :=[[-206.075578125,-38.1256328125,20.870232421875],[0.732123189175605,-0.57971865199821,0.222030212103854,-0.280400615744397],[0,0,0,0],[8.999999E+09,8.999999E+09,8.999999E+09,8.999999E+09,8.999999E+09,8.999999E+09]];
	LOCAL CONST Robtarget Tr_meulage_motif_1_P137 :=[[-205.304,-38.761765625,20.87033203125],[0.732123189175605,-0.57971865199821,0.222030212103854,-0.280400615744397],[0,0,0,0],[8.999999E+09,8.999999E+09,8.999999E+09,8.999999E+09,8.999999E+09,8.999999E+09]];
	LOCAL CONST Robtarget Tr_meulage_motif_1_P138 :=[[-204.532421875,-39.3978984375,20.8704296875],[0.732123189175605,-0.57971865199821,0.222030212103854,-0.280400615744397],[0,0,0,0],[8.999999E+09,8.999999E+09,8.999999E+09,8.999999E+09,8.999999E+09,8.999999E+09]];
	LOCAL CONST Robtarget Tr_meulage_motif_1_P139 :=[[-203.76084375,-40.03403125,20.870529296875],[0.732123189175605,-0.57971865199821,0.222030212103854,-0.280400615744397],[0,0,0,0],[8.999999E+09,8.999999E+09,8.999999E+09,8.999999E+09,8.999999E+09,8.999999E+09]];
	LOCAL CONST Robtarget Tr_meulage_motif_1_P140 :=[[-202.989265625,-40.6701640625,20.870626953125],[0.732123189175605,-0.57971865199821,0.222030212103854,-0.280400615744397],[0,0,0,0],[8.999999E+09,8.999999E+09,8.999999E+09,8.999999E+09,8.999999E+09,8.999999E+09]];
	LOCAL CONST Robtarget Tr_meulage_motif_1_P141 :=[[-202.2176875,-41.306296875,20.8707265625],[0.732123189175605,-0.57971865199821,0.222030212103854,-0.280400615744397],[0,0,0,0],[8.999999E+09,8.999999E+09,8.999999E+09,8.999999E+09,8.999999E+09,8.999999E+09]];
	LOCAL CONST Robtarget Tr_meulage_motif_1_P142 :=[[-201.44609375,-41.94243359375,20.87082421875],[0.732123189175605,-0.57971865199821,0.222030212103854,-0.280400615744397],[0,0,0,0],[8.999999E+09,8.999999E+09,8.999999E+09,8.999999E+09,8.999999E+09,8.999999E+09]];
	LOCAL CONST Robtarget Tr_meulage_motif_1_P143 :=[[-200.674515625,-42.57856640625,20.870921875],[0.732123189175605,-0.57971865199821,0.222030212103854,-0.280400615744397],[0,0,0,0],[8.999999E+09,8.999999E+09,8.999999E+09,8.999999E+09,8.999999E+09,8.999999E+09]];
	LOCAL CONST Robtarget Tr_meulage_motif_1_P144 :=[[-199.9029375,-43.21469921875,20.871021484375],[0.732123189175605,-0.57971865199821,0.222030212103854,-0.280400615744397],[0,0,0,0],[8.999999E+09,8.999999E+09,8.999999E+09,8.999999E+09,8.999999E+09,8.999999E+09]];
	LOCAL CONST Robtarget Tr_meulage_motif_1_P145 :=[[-199.131359375,-43.85083203125,20.871119140625],[0.732123189175605,-0.57971865199821,0.222030212103854,-0.280400615744397],[0,0,0,0],[8.999999E+09,8.999999E+09,8.999999E+09,8.999999E+09,8.999999E+09,8.999999E+09]];
	LOCAL CONST Robtarget Tr_meulage_motif_1_P146 :=[[-198.35978125,-44.48696484375,20.87121875],[0.732123189175605,-0.57971865199821,0.222030212103854,-0.280400615744397],[0,0,0,0],[8.999999E+09,8.999999E+09,8.999999E+09,8.999999E+09,8.999999E+09,8.999999E+09]];
	LOCAL CONST Robtarget Tr_meulage_motif_1_P147 :=[[-197.588203125,-45.12309765625,20.87131640625],[0.732123189175605,-0.57971865199821,0.222030212103854,-0.280400615744397],[0,0,0,0],[8.999999E+09,8.999999E+09,8.999999E+09,8.999999E+09,8.999999E+09,8.999999E+09]];
	LOCAL CONST Robtarget Tr_meulage_motif_1_P148 :=[[-196.816625,-45.75923046875,20.8714140625],[0.732123189175605,-0.57971865199821,0.222030212103854,-0.280400615744397],[0,0,0,0],[8.999999E+09,8.999999E+09,8.999999E+09,8.999999E+09,8.999999E+09,8.999999E+09]];
	LOCAL CONST Robtarget Tr_meulage_motif_1_P149 :=[[-196.045046875,-46.39536328125,20.871513671875],[0.732123189175605,-0.57971865199821,0.222030212103854,-0.280400615744397],[0,0,0,0],[8.999999E+09,8.999999E+09,8.999999E+09,8.999999E+09,8.999999E+09,8.999999E+09]];
	LOCAL CONST Robtarget Tr_meulage_motif_1_P150 :=[[-195.27346875,-47.03149609375,20.871611328125],[0.732123189175605,-0.57971865199821,0.222030212103854,-0.280400615744397],[0,0,0,0],[8.999999E+09,8.999999E+09,8.999999E+09,8.999999E+09,8.999999E+09,8.999999E+09]];
	LOCAL CONST Robtarget Tr_meulage_motif_1_P151 :=[[-194.501890625,-47.66762890625,20.8717109375],[0.732123189175605,-0.57971865199821,0.222030212103854,-0.280400615744397],[0,0,0,0],[8.999999E+09,8.999999E+09,8.999999E+09,8.999999E+09,8.999999E+09,8.999999E+09]];
	LOCAL CONST Robtarget Tr_meulage_motif_1_P152 :=[[-193.7303125,-48.303765625,20.87180859375],[0.732123189175605,-0.57971865199821,0.222030212103854,-0.280400615744397],[0,0,0,0],[8.999999E+09,8.999999E+09,8.999999E+09,8.999999E+09,8.999999E+09,8.999999E+09]];
	LOCAL CONST Robtarget Tr_meulage_motif_1_P153 :=[[-192.958734375,-48.9398984375,20.871908203125],[0.732123189175605,-0.57971865199821,0.222030212103854,-0.280400615744397],[0,0,0,0],[8.999999E+09,8.999999E+09,8.999999E+09,8.999999E+09,8.999999E+09,8.999999E+09]];
	LOCAL CONST Robtarget Tr_meulage_motif_1_P154 :=[[-192.18715625,-49.57603125,20.872005859375],[0.732123189175605,-0.57971865199821,0.222030212103854,-0.280400615744397],[0,0,0,0],[8.999999E+09,8.999999E+09,8.999999E+09,8.999999E+09,8.999999E+09,8.999999E+09]];
	LOCAL CONST Robtarget Tr_meulage_motif_1_P155 :=[[-191.415578125,-50.2121640625,20.872103515625],[0.732123189175605,-0.57971865199821,0.222030212103854,-0.280400615744397],[0,0,0,0],[8.999999E+09,8.999999E+09,8.999999E+09,8.999999E+09,8.999999E+09,8.999999E+09]];
	LOCAL CONST Robtarget Tr_meulage_motif_1_P156 :=[[-190.644,-50.848296875,20.872203125],[0.732123189175605,-0.57971865199821,0.222030212103854,-0.280400615744397],[0,0,0,0],[8.999999E+09,8.999999E+09,8.999999E+09,8.999999E+09,8.999999E+09,8.999999E+09]];
	LOCAL CONST Robtarget Tr_meulage_motif_1_P157 :=[[-189.87240625,-51.4844296875,20.87230078125],[0.732123189175605,-0.57971865199821,0.222030212103854,-0.280400615744397],[0,0,0,0],[8.999999E+09,8.999999E+09,8.999999E+09,8.999999E+09,8.999999E+09,8.999999E+09]];
	LOCAL CONST Robtarget Tr_meulage_motif_1_P158 :=[[-189.100828125,-52.1205625,20.872400390625],[0.732123189175605,-0.57971865199821,0.222030212103854,-0.280400615744397],[0,0,0,0],[8.999999E+09,8.999999E+09,8.999999E+09,8.999999E+09,8.999999E+09,8.999999E+09]];
	LOCAL CONST Robtarget Tr_meulage_motif_1_P159 :=[[-188.32925,-52.7566953125,20.872498046875],[0.732123189175605,-0.57971865199821,0.222030212103854,-0.280400615744397],[0,0,0,0],[8.999999E+09,8.999999E+09,8.999999E+09,8.999999E+09,8.999999E+09,8.999999E+09]];
	LOCAL CONST Robtarget Tr_meulage_motif_1_P160 :=[[-187.557671875,-53.392828125,20.872595703125],[0.732123189175605,-0.57971865199821,0.222030212103854,-0.280400615744397],[0,0,0,0],[8.999999E+09,8.999999E+09,8.999999E+09,8.999999E+09,8.999999E+09,8.999999E+09]];
	LOCAL CONST Robtarget Tr_meulage_motif_1_P161 :=[[-186.78609375,-54.02896484375,20.8726953125],[0.732123189175605,-0.57971865199821,0.222030212103854,-0.280400615744397],[0,0,0,0],[8.999999E+09,8.999999E+09,8.999999E+09,8.999999E+09,8.999999E+09,8.999999E+09]];
	LOCAL CONST Robtarget Tr_meulage_motif_1_P162 :=[[-186.014515625,-54.66509765625,20.87279296875],[0.732123189175605,-0.57971865199821,0.222030212103854,-0.280400615744397],[0,0,0,0],[8.999999E+09,8.999999E+09,8.999999E+09,8.999999E+09,8.999999E+09,8.999999E+09]];
	LOCAL CONST Robtarget Tr_meulage_motif_1_P163 :=[[-185.2429375,-55.30123046875,20.872892578125],[0.732123189175605,-0.57971865199821,0.222030212103854,-0.280400615744397],[0,0,0,0],[8.999999E+09,8.999999E+09,8.999999E+09,8.999999E+09,8.999999E+09,8.999999E+09]];
	LOCAL CONST Robtarget Tr_meulage_motif_1_P164 :=[[-184.471359375,-55.93736328125,20.872990234375],[0.732123189175605,-0.57971865199821,0.222030212103854,-0.280400615744397],[0,0,0,0],[8.999999E+09,8.999999E+09,8.999999E+09,8.999999E+09,8.999999E+09,8.999999E+09]];
	LOCAL CONST Robtarget Tr_meulage_motif_1_P165 :=[[-183.69978125,-56.57349609375,20.87308984375],[0.732123189175605,-0.57971865199821,0.222030212103854,-0.280400615744397],[0,0,0,0],[8.999999E+09,8.999999E+09,8.999999E+09,8.999999E+09,8.999999E+09,8.999999E+09]];
	LOCAL CONST Robtarget Tr_meulage_motif_1_P166 :=[[-182.928203125,-57.20962890625,20.8731875],[0.732123189175605,-0.57971865199821,0.222030212103854,-0.280400615744397],[0,0,0,0],[8.999999E+09,8.999999E+09,8.999999E+09,8.999999E+09,8.999999E+09,8.999999E+09]];
	LOCAL CONST Robtarget Tr_meulage_motif_1_P167 :=[[-182.156625,-57.84576171875,20.87328515625],[0.732123189175605,-0.57971865199821,0.222030212103854,-0.280400615744397],[0,0,0,0],[8.999999E+09,8.999999E+09,8.999999E+09,8.999999E+09,8.999999E+09,8.999999E+09]];
	LOCAL CONST Robtarget Tr_meulage_motif_1_P168 :=[[-181.385046875,-58.48189453125,20.873384765625],[0.732123189175605,-0.57971865199821,0.222030212103854,-0.280400615744397],[0,0,0,0],[8.999999E+09,8.999999E+09,8.999999E+09,8.999999E+09,8.999999E+09,8.999999E+09]];
	LOCAL CONST Robtarget Tr_meulage_motif_1_P169 :=[[-180.61346875,-59.11802734375,20.873482421875],[0.732123189175605,-0.57971865199821,0.222030212103854,-0.280400615744397],[0,0,0,0],[8.999999E+09,8.999999E+09,8.999999E+09,8.999999E+09,8.999999E+09,8.999999E+09]];
	LOCAL CONST Robtarget Tr_meulage_motif_1_P170 :=[[-179.841890625,-59.75416015625,20.87358203125],[0.732123189175605,-0.57971865199821,0.222030212103854,-0.280400615744397],[0,0,0,0],[8.999999E+09,8.999999E+09,8.999999E+09,8.999999E+09,8.999999E+09,8.999999E+09]];
	LOCAL CONST Robtarget Tr_meulage_motif_1_P171 :=[[-179.070296875,-60.390296875,20.8736796875],[0.732123189175605,-0.57971865199821,0.222030212103854,-0.280400615744397],[0,0,0,0],[8.999999E+09,8.999999E+09,8.999999E+09,8.999999E+09,8.999999E+09,8.999999E+09]];
	LOCAL CONST Robtarget Tr_meulage_motif_1_P172 :=[[-178.29871875,-61.0264296875,20.873779296875],[0.732123189175605,-0.57971865199821,0.222030212103854,-0.280400615744397],[0,0,0,0],[8.999999E+09,8.999999E+09,8.999999E+09,8.999999E+09,8.999999E+09,8.999999E+09]];
	LOCAL CONST Robtarget Tr_meulage_motif_1_P173 :=[[-177.527140625,-61.6625625,20.873876953125],[0.732123189175605,-0.57971865199821,0.222030212103854,-0.280400615744397],[0,0,0,0],[8.999999E+09,8.999999E+09,8.999999E+09,8.999999E+09,8.999999E+09,8.999999E+09]];
	LOCAL CONST Robtarget Tr_meulage_motif_1_P174 :=[[-176.757421875,-62.28926953125,20.763548828125],[0.732123189175605,-0.57971865199821,0.222030212103854,-0.280400615744397],[0,0,0,0],[8.999999E+09,8.999999E+09,8.999999E+09,8.999999E+09,8.999999E+09,8.999999E+09]];
	LOCAL CONST Robtarget Tr_meulage_motif_1_P175 :=[[-176.019703125,-62.88240625,20.552775390625],[0.732123189175605,-0.57971865199821,0.222030212103854,-0.280400615744397],[0,0,0,0],[8.999999E+09,8.999999E+09,8.999999E+09,8.999999E+09,8.999999E+09,8.999999E+09]];
	LOCAL CONST Robtarget Tr_meulage_motif_1_P176 :=[[-175.35221875,-63.41331640625,20.281427734375],[0.732123189175605,-0.57971865199821,0.222030212103854,-0.280400615744397],[0,0,0,0],[8.999999E+09,8.999999E+09,8.999999E+09,8.999999E+09,8.999999E+09,8.999999E+09]];
	LOCAL CONST Robtarget Tr_meulage_motif_1_P177 :=[[-174.763890625,-63.8786640625,20.005982421875],[0.732123189175605,-0.57971865199821,0.222030212103854,-0.280400615744397],[0,0,0,0],[8.999999E+09,8.999999E+09,8.999999E+09,8.999999E+09,8.999999E+09,8.999999E+09]];
	LOCAL CONST Robtarget Tr_meulage_motif_1_P178 :=[[-173.892703125,-64.55294140625,19.39090234375],[0.732123189175605,-0.57971865199821,0.222030212103854,-0.280400615744397],[0,0,0,0],[8.999999E+09,8.999999E+09,8.999999E+09,8.999999E+09,8.999999E+09,8.999999E+09]];
	LOCAL CONST Robtarget Tr_meulage_motif_1_P179 :=[[-173.0729375,-65.1682890625,18.5446328125],[0.732123189175605,-0.57971865199821,0.222030212103854,-0.280400615744397],[0,0,0,0],[8.999999E+09,8.999999E+09,8.999999E+09,8.999999E+09,8.999999E+09,8.999999E+09]];
	LOCAL CONST Robtarget Tr_meulage_motif_1_P180 :=[[-172.382953125,-65.6640625,17.522396484375],[0.732123189175605,-0.57971865199821,0.222030212103854,-0.280400615744397],[0,0,0,0],[8.999999E+09,8.999999E+09,8.999999E+09,8.999999E+09,8.999999E+09,8.999999E+09]];
	LOCAL CONST Robtarget Tr_meulage_motif_1_P181 :=[[-171.96709375,-65.9272265625,16.407951171875],[0.732123189175605,-0.57971865199821,0.222030212103854,-0.280400615744397],[0,0,0,0],[8.999999E+09,8.999999E+09,8.999999E+09,8.999999E+09,8.999999E+09,8.999999E+09]];
	LOCAL CONST Robtarget Tr_meulage_motif_1_P182 :=[[-171.92178125,-65.91490625,15.7130419921875],[0.732123189175605,-0.57971865199821,0.222030212103854,-0.280400615744397],[0,0,0,0],[8.999999E+09,8.999999E+09,8.999999E+09,8.999999E+09,8.999999E+09,8.999999E+09]];
	LOCAL CONST Robtarget Tr_meulage_motif_1_P183 :=[[-171.8985625,-65.88684375,15.0527958984375],[0.732123189175605,-0.57971865199821,0.222030212103854,-0.280400615744397],[0,0,0,0],[8.999999E+09,8.999999E+09,8.999999E+09,8.999999E+09,8.999999E+09,8.999999E+09]];
	LOCAL CONST Robtarget Tr_meulage_motif_1_P184 :=[[-171.9176875,-65.8238828125,14.3927001953125],[0.732123189175605,-0.57971865199821,0.222030212103854,-0.280400615744397],[0,0,0,0],[8.999999E+09,8.999999E+09,8.999999E+09,8.999999E+09,8.999999E+09,8.999999E+09]];
	LOCAL CONST Robtarget Tr_meulage_motif_1_P185 :=[[-172.263421875,-65.46019140625,13.29257421875],[0.732123189175605,-0.57971865199821,0.222030212103854,-0.280400615744397],[0,0,0,0],[8.999999E+09,8.999999E+09,8.999999E+09,8.999999E+09,8.999999E+09,8.999999E+09]];
	LOCAL CONST Robtarget Tr_meulage_motif_1_P186 :=[[-172.889015625,-64.872546875,12.287392578125],[0.732123189175605,-0.57971865199821,0.222030212103854,-0.280400615744397],[0,0,0,0],[8.999999E+09,8.999999E+09,8.999999E+09,8.999999E+09,8.999999E+09,8.999999E+09]];
	LOCAL CONST Robtarget Tr_meulage_motif_1_P187 :=[[-173.649546875,-64.18634765625,11.45967578125],[0.732123189175605,-0.57971865199821,0.222030212103854,-0.280400615744397],[0,0,0,0],[8.999999E+09,8.999999E+09,8.999999E+09,8.999999E+09,8.999999E+09,8.999999E+09]];
	LOCAL CONST Robtarget Tr_meulage_motif_1_P188 :=[[-174.165796875,-63.73246875,11.0644580078125],[0.732123189175605,-0.57971865199821,0.222030212103854,-0.280400615744397],[0,0,0,0],[8.999999E+09,8.999999E+09,8.999999E+09,8.999999E+09,8.999999E+09,8.999999E+09]];
	LOCAL CONST Robtarget Tr_meulage_motif_1_P189 :=[[-175.042296875,-62.9750390625,10.5775537109375],[0.732123189175605,-0.57971865199821,0.222030212103854,-0.280400615744397],[0,0,0,0],[8.999999E+09,8.999999E+09,8.999999E+09,8.999999E+09,8.999999E+09,8.999999E+09]];
	LOCAL CONST Robtarget Tr_meulage_motif_1_P190 :=[[-175.68503125,-62.42627734375,10.31377734375],[0.732123189175605,-0.57971865199821,0.222030212103854,-0.280400615744397],[0,0,0,0],[8.999999E+09,8.999999E+09,8.999999E+09,8.999999E+09,8.999999E+09,8.999999E+09]];
	LOCAL CONST Robtarget Tr_meulage_motif_1_P191 :=[[-176.396953125,-61.8247265625,10.10952734375],[0.732123189175605,-0.57971865199821,0.222030212103854,-0.280400615744397],[0,0,0,0],[8.999999E+09,8.999999E+09,8.999999E+09,8.999999E+09,8.999999E+09,8.999999E+09]];
	LOCAL CONST Robtarget Tr_meulage_motif_1_P192 :=[[-177.1505,-61.1957109375,10.001001953125],[0.732123189175605,-0.57971865199821,0.222030212103854,-0.280400615744397],[0,0,0,0],[8.999999E+09,8.999999E+09,8.999999E+09,8.999999E+09,8.999999E+09,8.999999E+09]];
	LOCAL CONST Robtarget Tr_meulage_motif_1_P193 :=[[-177.912453125,-60.5596171875,9.890478515625],[0.732123189175605,-0.57971865199821,0.222030212103854,-0.280400615744397],[0,0,0,0],[8.999999E+09,8.999999E+09,8.999999E+09,8.999999E+09,8.999999E+09,8.999999E+09]];
	LOCAL CONST Robtarget Tr_meulage_motif_1_P194 :=[[-178.68403125,-59.923484375,9.8903798828125],[0.732123189175605,-0.57971865199821,0.222030212103854,-0.280400615744397],[0,0,0,0],[8.999999E+09,8.999999E+09,8.999999E+09,8.999999E+09,8.999999E+09,8.999999E+09]];
	LOCAL CONST Robtarget Tr_meulage_motif_1_P195 :=[[-179.455609375,-59.2873515625,9.89028125],[0.732123189175605,-0.57971865199821,0.222030212103854,-0.280400615744397],[0,0,0,0],[8.999999E+09,8.999999E+09,8.999999E+09,8.999999E+09,8.999999E+09,8.999999E+09]];
	LOCAL CONST Robtarget Tr_meulage_motif_1_P196 :=[[-180.2271875,-58.65121875,9.8901826171875],[0.732123189175605,-0.57971865199821,0.222030212103854,-0.280400615744397],[0,0,0,0],[8.999999E+09,8.999999E+09,8.999999E+09,8.999999E+09,8.999999E+09,8.999999E+09]];
	LOCAL CONST Robtarget Tr_meulage_motif_1_P197 :=[[-180.99878125,-58.0150859375,9.890083984375],[0.732123189175605,-0.57971865199821,0.222030212103854,-0.280400615744397],[0,0,0,0],[8.999999E+09,8.999999E+09,8.999999E+09,8.999999E+09,8.999999E+09,8.999999E+09]];
	LOCAL CONST Robtarget Tr_meulage_motif_1_P198 :=[[-181.770359375,-57.37894921875,9.8899853515625],[0.732123189175605,-0.57971865199821,0.222030212103854,-0.280400615744397],[0,0,0,0],[8.999999E+09,8.999999E+09,8.999999E+09,8.999999E+09,8.999999E+09,8.999999E+09]];
	LOCAL CONST Robtarget Tr_meulage_motif_1_P199 :=[[-182.5419375,-56.74281640625,9.8898876953125],[0.732123189175605,-0.57971865199821,0.222030212103854,-0.280400615744397],[0,0,0,0],[8.999999E+09,8.999999E+09,8.999999E+09,8.999999E+09,8.999999E+09,8.999999E+09]];
	LOCAL CONST Robtarget Tr_meulage_motif_1_P200 :=[[-183.313515625,-56.10668359375,9.8897890625],[0.732123189175605,-0.57971865199821,0.222030212103854,-0.280400615744397],[0,0,0,0],[8.999999E+09,8.999999E+09,8.999999E+09,8.999999E+09,8.999999E+09,8.999999E+09]];
	LOCAL CONST Robtarget Tr_meulage_motif_1_P201 :=[[-184.08509375,-55.47055078125,9.8896904296875],[0.732123189175605,-0.57971865199821,0.222030212103854,-0.280400615744397],[0,0,0,0],[8.999999E+09,8.999999E+09,8.999999E+09,8.999999E+09,8.999999E+09,8.999999E+09]];
	LOCAL CONST Robtarget Tr_meulage_motif_1_P202 :=[[-184.856671875,-54.83441796875,9.889591796875],[0.732123189175605,-0.57971865199821,0.222030212103854,-0.280400615744397],[0,0,0,0],[8.999999E+09,8.999999E+09,8.999999E+09,8.999999E+09,8.999999E+09,8.999999E+09]];
	LOCAL CONST Robtarget Tr_meulage_motif_1_P203 :=[[-185.62825,-54.19828515625,9.8894931640625],[0.732123189175605,-0.57971865199821,0.222030212103854,-0.280400615744397],[0,0,0,0],[8.999999E+09,8.999999E+09,8.999999E+09,8.999999E+09,8.999999E+09,8.999999E+09]];
	LOCAL CONST Robtarget Tr_meulage_motif_1_P204 :=[[-186.399828125,-53.56215234375,9.88939453125],[0.732123189175605,-0.57971865199821,0.222030212103854,-0.280400615744397],[0,0,0,0],[8.999999E+09,8.999999E+09,8.999999E+09,8.999999E+09,8.999999E+09,8.999999E+09]];
	LOCAL CONST Robtarget Tr_meulage_motif_1_P205 :=[[-187.17140625,-52.92601953125,9.889296875],[0.732123189175605,-0.57971865199821,0.222030212103854,-0.280400615744397],[0,0,0,0],[8.999999E+09,8.999999E+09,8.999999E+09,8.999999E+09,8.999999E+09,8.999999E+09]];
	LOCAL CONST Robtarget Tr_meulage_motif_1_P206 :=[[-187.942984375,-52.28988671875,9.8891982421875],[0.732123189175605,-0.57971865199821,0.222030212103854,-0.280400615744397],[0,0,0,0],[8.999999E+09,8.999999E+09,8.999999E+09,8.999999E+09,8.999999E+09,8.999999E+09]];
	LOCAL CONST Robtarget Tr_meulage_motif_1_P207 :=[[-188.7145625,-51.65375,9.889099609375],[0.732123189175605,-0.57971865199821,0.222030212103854,-0.280400615744397],[0,0,0,0],[8.999999E+09,8.999999E+09,8.999999E+09,8.999999E+09,8.999999E+09,8.999999E+09]];
	LOCAL CONST Robtarget Tr_meulage_motif_1_P208 :=[[-189.486140625,-51.0176171875,9.8890009765625],[0.732123189175605,-0.57971865199821,0.222030212103854,-0.280400615744397],[0,0,0,0],[8.999999E+09,8.999999E+09,8.999999E+09,8.999999E+09,8.999999E+09,8.999999E+09]];
	LOCAL CONST Robtarget Tr_meulage_motif_1_P209 :=[[-190.25771875,-50.381484375,9.88890234375],[0.732123189175605,-0.57971865199821,0.222030212103854,-0.280400615744397],[0,0,0,0],[8.999999E+09,8.999999E+09,8.999999E+09,8.999999E+09,8.999999E+09,8.999999E+09]];
	LOCAL CONST Robtarget Tr_meulage_motif_1_P210 :=[[-191.029296875,-49.7453515625,9.8888037109375],[0.732123189175605,-0.57971865199821,0.222030212103854,-0.280400615744397],[0,0,0,0],[8.999999E+09,8.999999E+09,8.999999E+09,8.999999E+09,8.999999E+09,8.999999E+09]];
	LOCAL CONST Robtarget Tr_meulage_motif_1_P211 :=[[-191.800890625,-49.10921875,9.888705078125],[0.732123189175605,-0.57971865199821,0.222030212103854,-0.280400615744397],[0,0,0,0],[8.999999E+09,8.999999E+09,8.999999E+09,8.999999E+09,8.999999E+09,8.999999E+09]];
	LOCAL CONST Robtarget Tr_meulage_motif_1_P212 :=[[-192.57246875,-48.4730859375,9.888607421875],[0.732123189175605,-0.57971865199821,0.222030212103854,-0.280400615744397],[0,0,0,0],[8.999999E+09,8.999999E+09,8.999999E+09,8.999999E+09,8.999999E+09,8.999999E+09]];
	LOCAL CONST Robtarget Tr_meulage_motif_1_P213 :=[[-193.344046875,-47.836953125,9.8885087890625],[0.732123189175605,-0.57971865199821,0.222030212103854,-0.280400615744397],[0,0,0,0],[8.999999E+09,8.999999E+09,8.999999E+09,8.999999E+09,8.999999E+09,8.999999E+09]];
	LOCAL CONST Robtarget Tr_meulage_motif_1_P214 :=[[-194.115625,-47.2008203125,9.88841015625],[0.732123189175605,-0.57971865199821,0.222030212103854,-0.280400615744397],[0,0,0,0],[8.999999E+09,8.999999E+09,8.999999E+09,8.999999E+09,8.999999E+09,8.999999E+09]];
	LOCAL CONST Robtarget Tr_meulage_motif_1_P215 :=[[-194.887203125,-46.5646875,9.8883115234375],[0.732123189175605,-0.57971865199821,0.222030212103854,-0.280400615744397],[0,0,0,0],[8.999999E+09,8.999999E+09,8.999999E+09,8.999999E+09,8.999999E+09,8.999999E+09]];
	LOCAL CONST Robtarget Tr_meulage_motif_1_P216 :=[[-195.65878125,-45.9285546875,9.888212890625],[0.732123189175605,-0.57971865199821,0.222030212103854,-0.280400615744397],[0,0,0,0],[8.999999E+09,8.999999E+09,8.999999E+09,8.999999E+09,8.999999E+09,8.999999E+09]];
	LOCAL CONST Robtarget Tr_meulage_motif_1_P217 :=[[-196.430359375,-45.29241796875,9.8881142578125],[0.732123189175605,-0.57971865199821,0.222030212103854,-0.280400615744397],[0,0,0,0],[8.999999E+09,8.999999E+09,8.999999E+09,8.999999E+09,8.999999E+09,8.999999E+09]];
	LOCAL CONST Robtarget Tr_meulage_motif_1_P218 :=[[-197.2019375,-44.65628515625,9.8880166015625],[0.732123189175605,-0.57971865199821,0.222030212103854,-0.280400615744397],[0,0,0,0],[8.999999E+09,8.999999E+09,8.999999E+09,8.999999E+09,8.999999E+09,8.999999E+09]];
	LOCAL CONST Robtarget Tr_meulage_motif_1_P219 :=[[-197.973515625,-44.02015234375,9.88791796875],[0.732123189175605,-0.57971865199821,0.222030212103854,-0.280400615744397],[0,0,0,0],[8.999999E+09,8.999999E+09,8.999999E+09,8.999999E+09,8.999999E+09,8.999999E+09]];
	LOCAL CONST Robtarget Tr_meulage_motif_1_P220 :=[[-198.74509375,-43.38401953125,9.8878193359375],[0.732123189175605,-0.57971865199821,0.222030212103854,-0.280400615744397],[0,0,0,0],[8.999999E+09,8.999999E+09,8.999999E+09,8.999999E+09,8.999999E+09,8.999999E+09]];
	LOCAL CONST Robtarget Tr_meulage_motif_1_P221 :=[[-199.516671875,-42.74788671875,9.887720703125],[0.732123189175605,-0.57971865199821,0.222030212103854,-0.280400615744397],[0,0,0,0],[8.999999E+09,8.999999E+09,8.999999E+09,8.999999E+09,8.999999E+09,8.999999E+09]];
	LOCAL CONST Robtarget Tr_meulage_motif_1_P222 :=[[-200.28825,-42.11175390625,9.8876220703125],[0.732123189175605,-0.57971865199821,0.222030212103854,-0.280400615744397],[0,0,0,0],[8.999999E+09,8.999999E+09,8.999999E+09,8.999999E+09,8.999999E+09,8.999999E+09]];
	LOCAL CONST Robtarget Tr_meulage_motif_1_P223 :=[[-201.059828125,-41.47562109375,9.8875234375],[0.732123189175605,-0.57971865199821,0.222030212103854,-0.280400615744397],[0,0,0,0],[8.999999E+09,8.999999E+09,8.999999E+09,8.999999E+09,8.999999E+09,8.999999E+09]];
	LOCAL CONST Robtarget Tr_meulage_motif_1_P224 :=[[-201.83140625,-40.83948828125,9.88742578125],[0.732123189175605,-0.57971865199821,0.222030212103854,-0.280400615744397],[0,0,0,0],[8.999999E+09,8.999999E+09,8.999999E+09,8.999999E+09,8.999999E+09,8.999999E+09]];
	LOCAL CONST Robtarget Tr_meulage_motif_1_P225 :=[[-202.603,-40.20335546875,9.8873271484375],[0.732123189175605,-0.57971865199821,0.222030212103854,-0.280400615744397],[0,0,0,0],[8.999999E+09,8.999999E+09,8.999999E+09,8.999999E+09,8.999999E+09,8.999999E+09]];
	LOCAL CONST Robtarget Tr_meulage_motif_1_P226 :=[[-203.374578125,-39.56721875,9.887228515625],[0.732123189175605,-0.57971865199821,0.222030212103854,-0.280400615744397],[0,0,0,0],[8.999999E+09,8.999999E+09,8.999999E+09,8.999999E+09,8.999999E+09,8.999999E+09]];
	LOCAL CONST Robtarget Tr_meulage_motif_1_P227 :=[[-204.14615625,-38.9310859375,9.8871298828125],[0.732123189175605,-0.57971865199821,0.222030212103854,-0.280400615744397],[0,0,0,0],[8.999999E+09,8.999999E+09,8.999999E+09,8.999999E+09,8.999999E+09,8.999999E+09]];
	LOCAL CONST Robtarget Tr_meulage_motif_1_P228 :=[[-204.917734375,-38.294953125,9.88703125],[0.732123189175605,-0.57971865199821,0.222030212103854,-0.280400615744397],[0,0,0,0],[8.999999E+09,8.999999E+09,8.999999E+09,8.999999E+09,8.999999E+09,8.999999E+09]];
	LOCAL CONST Robtarget Tr_meulage_motif_1_P229 :=[[-205.6893125,-37.6588203125,9.8869326171875],[0.732123189175605,-0.57971865199821,0.222030212103854,-0.280400615744397],[0,0,0,0],[8.999999E+09,8.999999E+09,8.999999E+09,8.999999E+09,8.999999E+09,8.999999E+09]];
	LOCAL CONST Robtarget Tr_meulage_motif_1_P230 :=[[-206.460890625,-37.0226875,9.8868349609375],[0.732123189175605,-0.57971865199821,0.222030212103854,-0.280400615744397],[0,0,0,0],[8.999999E+09,8.999999E+09,8.999999E+09,8.999999E+09,8.999999E+09,8.999999E+09]];
	LOCAL CONST Robtarget Tr_meulage_motif_1_P231 :=[[-207.23246875,-36.3865546875,9.886736328125],[0.732123189175605,-0.57971865199821,0.222030212103854,-0.280400615744397],[0,0,0,0],[8.999999E+09,8.999999E+09,8.999999E+09,8.999999E+09,8.999999E+09,8.999999E+09]];
	LOCAL CONST Robtarget Tr_meulage_motif_1_P232 :=[[-208.004046875,-35.750421875,9.8866376953125],[0.732123189175605,-0.57971865199821,0.222030212103854,-0.280400615744397],[0,0,0,0],[8.999999E+09,8.999999E+09,8.999999E+09,8.999999E+09,8.999999E+09,8.999999E+09]];
	LOCAL CONST Robtarget Tr_meulage_motif_1_P233 :=[[-208.775625,-35.1142890625,9.8865390625],[0.732123189175605,-0.57971865199821,0.222030212103854,-0.280400615744397],[0,0,0,0],[8.999999E+09,8.999999E+09,8.999999E+09,8.999999E+09,8.999999E+09,8.999999E+09]];
	LOCAL CONST Robtarget Tr_meulage_motif_1_P234 :=[[-209.547203125,-34.47815625,9.8864404296875],[0.732123189175605,-0.57971865199821,0.222030212103854,-0.280400615744397],[0,0,0,0],[8.999999E+09,8.999999E+09,8.999999E+09,8.999999E+09,8.999999E+09,8.999999E+09]];
	LOCAL CONST Robtarget Tr_meulage_motif_1_P235 :=[[-210.31878125,-33.8420234375,9.886341796875],[0.732123189175605,-0.57971865199821,0.222030212103854,-0.280400615744397],[0,0,0,0],[8.999999E+09,8.999999E+09,8.999999E+09,8.999999E+09,8.999999E+09,8.999999E+09]];
	LOCAL CONST Robtarget Tr_meulage_motif_1_P236 :=[[-211.080734375,-33.20592578125,9.775818359375],[0.732123189175605,-0.57971865199821,0.222030212103854,-0.280400615744397],[0,0,0,0],[8.999999E+09,8.999999E+09,8.999999E+09,8.999999E+09,8.999999E+09,8.999999E+09]];
	LOCAL CONST Robtarget Tr_meulage_motif_1_P237 :=[[-211.803625,-32.59486328125,9.5648583984375],[0.732123189175605,-0.57971865199821,0.222030212103854,-0.280400615744397],[0,0,0,0],[8.999999E+09,8.999999E+09,8.999999E+09,8.999999E+09,8.999999E+09,8.999999E+09]];
	LOCAL CONST Robtarget Tr_meulage_motif_1_P238 :=[[-212.452015625,-32.040884765625,9.29334375],[0.732123189175605,-0.57971865199821,0.222030212103854,-0.280400615744397],[0,0,0,0],[8.999999E+09,8.999999E+09,8.999999E+09,8.999999E+09,8.999999E+09,8.999999E+09]];
	LOCAL CONST Robtarget Tr_meulage_motif_1_P239 :=[[-212.9903125,-31.575369140625,8.9895947265625],[0.732123189175605,-0.57971865199821,0.222030212103854,-0.280400615744397],[0,0,0,0],[8.999999E+09,8.999999E+09,8.999999E+09,8.999999E+09,8.999999E+09,8.999999E+09]];
	LOCAL CONST Robtarget Tr_meulage_motif_1_P240 :=[[-213.765234375,-30.889193359375,8.3279677734375],[0.732123189175605,-0.57971865199821,0.222030212103854,-0.280400615744397],[0,0,0,0],[8.999999E+09,8.999999E+09,8.999999E+09,8.999999E+09,8.999999E+09,8.999999E+09]];
	LOCAL CONST Robtarget Tr_meulage_motif_1_P241 :=[[-214.42946875,-30.2771640625,7.42729443359375],[0.732123189175605,-0.57971865199821,0.222030212103854,-0.280400615744397],[0,0,0,0],[8.999999E+09,8.999999E+09,8.999999E+09,8.999999E+09,8.999999E+09,8.999999E+09]];
	LOCAL CONST Robtarget Tr_meulage_motif_1_P242 :=[[-214.805515625,-29.892462890625,6.382814453125],[0.732123189175605,-0.57971865199821,0.222030212103854,-0.280400615744397],[0,0,0,0],[8.999999E+09,8.999999E+09,8.999999E+09,8.999999E+09,8.999999E+09,8.999999E+09]];
	LOCAL CONST Robtarget Tr_meulage_motif_1_P243 :=[[-214.92375,-29.745498046875,5.6906142578125],[0.732123189175605,-0.57971865199821,0.222030212103854,-0.280400615744397],[0,0,0,0],[8.999999E+09,8.999999E+09,8.999999E+09,8.999999E+09,8.999999E+09,8.999999E+09]];
	LOCAL CONST Robtarget Tr_meulage_motif_1_P244 :=[[-214.94596875,-29.672208984375,4.92177685546875],[0.732123189175605,-0.57971865199821,0.222030212103854,-0.280400615744397],[0,0,0,0],[8.999999E+09,8.999999E+09,8.999999E+09,8.999999E+09,8.999999E+09,8.999999E+09]];
	LOCAL CONST Robtarget Tr_meulage_motif_1_P245 :=[[-214.86728125,-29.682119140625,4.1530927734375],[0.732123189175605,-0.57971865199821,0.222030212103854,-0.280400615744397],[0,0,0,0],[8.999999E+09,8.999999E+09,8.999999E+09,8.999999E+09,8.999999E+09,8.999999E+09]];
	LOCAL CONST Robtarget Tr_meulage_motif_1_P246 :=[[-214.504609375,-29.90200390625,3.04656665039063],[0.732123189175605,-0.57971865199821,0.222030212103854,-0.280400615744397],[0,0,0,0],[8.999999E+09,8.999999E+09,8.999999E+09,8.999999E+09,8.999999E+09,8.999999E+09]];
	LOCAL CONST Robtarget Tr_meulage_motif_1_P247 :=[[-214.164375,-30.14070703125,2.46180908203125],[0.732123189175605,-0.57971865199821,0.222030212103854,-0.280400615744397],[0,0,0,0],[8.999999E+09,8.999999E+09,8.999999E+09,8.999999E+09,8.999999E+09,8.999999E+09]];
	LOCAL CONST Robtarget Tr_meulage_motif_1_P248 :=[[-213.448734375,-30.667388671875,1.57608715820313],[0.732123189175605,-0.57971865199821,0.222030212103854,-0.280400615744397],[0,0,0,0],[8.999999E+09,8.999999E+09,8.999999E+09,8.999999E+09,8.999999E+09,8.999999E+09]];
	LOCAL CONST Robtarget Tr_meulage_motif_1_P249 :=[[-212.98228125,-31.0223828125,1.16249255371094],[0.732123189175605,-0.57971865199821,0.222030212103854,-0.280400615744397],[0,0,0,0],[8.999999E+09,8.999999E+09,8.999999E+09,8.999999E+09,8.999999E+09,8.999999E+09]];
	LOCAL CONST Robtarget Tr_meulage_motif_1_P250 :=[[-212.100625,-31.7104296875,0.619303649902344],[0.732123189175605,-0.57971865199821,0.222030212103854,-0.280400615744397],[0,0,0,0],[8.999999E+09,8.999999E+09,8.999999E+09,8.999999E+09,8.999999E+09,8.999999E+09]];
	LOCAL CONST Robtarget Tr_meulage_motif_1_P251 :=[[-211.453234375,-32.223076171875,0.324333587646484],[0.732123189175605,-0.57971865199821,0.222030212103854,-0.280400615744397],[0,0,0,0],[8.999999E+09,8.999999E+09,8.999999E+09,8.999999E+09,8.999999E+09,8.999999E+09]];
	LOCAL CONST Robtarget Tr_meulage_motif_1_P252 :=[[-210.7269375,-32.8072734375,0.120251419067383],[0.732123189175605,-0.57971865199821,0.222030212103854,-0.280400615744397],[0,0,0,0],[8.999999E+09,8.999999E+09,8.999999E+09,8.999999E+09,8.999999E+09,8.999999E+09]];
	LOCAL CONST Robtarget Tr_meulage_motif_1_P253 :=[[-209.96578125,-33.42707421875,0.0119659957885742],[0.732123189175605,-0.57971865199821,0.222030212103854,-0.280400615744397],[0,0,0,0],[8.999999E+09,8.999999E+09,8.999999E+09,8.999999E+09,8.999999E+09,8.999999E+09]];
	LOCAL CONST Robtarget Tr_meulage_motif_1_P254 :=[[-209.196046875,-34.05378125,-0.0983777160644531],[0.732123189175605,-0.57971865199821,0.222030212103854,-0.280400615744397],[0,0,0,0],[8.999999E+09,8.999999E+09,8.999999E+09,8.999999E+09,8.999999E+09,8.999999E+09]];
	LOCAL CONST Robtarget Tr_meulage_motif_1_P255 :=[[-208.42446875,-34.6899140625,-0.0982792434692383],[0.732123189175605,-0.57971865199821,0.222030212103854,-0.280400615744397],[0,0,0,0],[8.999999E+09,8.999999E+09,8.999999E+09,8.999999E+09,8.999999E+09,8.999999E+09]];
	LOCAL CONST Robtarget Tr_meulage_motif_1_P256 :=[[-207.652890625,-35.326046875,-0.0981807708740234],[0.732123189175605,-0.57971865199821,0.222030212103854,-0.280400615744397],[0,0,0,0],[8.999999E+09,8.999999E+09,8.999999E+09,8.999999E+09,8.999999E+09,8.999999E+09]];
	LOCAL CONST Robtarget Tr_meulage_motif_1_P257 :=[[-206.8813125,-35.9621796875,-0.0980822982788086],[0.732123189175605,-0.57971865199821,0.222030212103854,-0.280400615744397],[0,0,0,0],[8.999999E+09,8.999999E+09,8.999999E+09,8.999999E+09,8.999999E+09,8.999999E+09]];
	LOCAL CONST Robtarget Tr_meulage_motif_1_P258 :=[[-206.109734375,-36.5983125,-0.0979838256835937],[0.732123189175605,-0.57971865199821,0.222030212103854,-0.280400615744397],[0,0,0,0],[8.999999E+09,8.999999E+09,8.999999E+09,8.999999E+09,8.999999E+09,8.999999E+09]];
	LOCAL CONST Robtarget Tr_meulage_motif_1_P259 :=[[-205.33815625,-37.2344453125,-0.0978853530883789],[0.732123189175605,-0.57971865199821,0.222030212103854,-0.280400615744397],[0,0,0,0],[8.999999E+09,8.999999E+09,8.999999E+09,8.999999E+09,8.999999E+09,8.999999E+09]];
	LOCAL CONST Robtarget Tr_meulage_motif_1_P260 :=[[-204.566578125,-37.87058203125,-0.0977868804931641],[0.732123189175605,-0.57971865199821,0.222030212103854,-0.280400615744397],[0,0,0,0],[8.999999E+09,8.999999E+09,8.999999E+09,8.999999E+09,8.999999E+09,8.999999E+09]];
	LOCAL CONST Robtarget Tr_meulage_motif_1_P261 :=[[-203.795,-38.50671484375,-0.0976884078979492],[0.732123189175605,-0.57971865199821,0.222030212103854,-0.280400615744397],[0,0,0,0],[8.999999E+09,8.999999E+09,8.999999E+09,8.999999E+09,8.999999E+09,8.999999E+09]];
	LOCAL CONST Robtarget Tr_meulage_motif_1_P262 :=[[-203.023421875,-39.14284765625,-0.0975899353027344],[0.732123189175605,-0.57971865199821,0.222030212103854,-0.280400615744397],[0,0,0,0],[8.999999E+09,8.999999E+09,8.999999E+09,8.999999E+09,8.999999E+09,8.999999E+09]];
	LOCAL CONST Robtarget Tr_meulage_motif_1_P263 :=[[-202.25184375,-39.77898046875,-0.0974914703369141],[0.732123189175605,-0.57971865199821,0.222030212103854,-0.280400615744397],[0,0,0,0],[8.999999E+09,8.999999E+09,8.999999E+09,8.999999E+09,8.999999E+09,8.999999E+09]];
	LOCAL CONST Robtarget Tr_meulage_motif_1_P264 :=[[-201.480265625,-40.41511328125,-0.0973929977416992],[0.732123189175605,-0.57971865199821,0.222030212103854,-0.280400615744397],[0,0,0,0],[8.999999E+09,8.999999E+09,8.999999E+09,8.999999E+09,8.999999E+09,8.999999E+09]];
	LOCAL CONST Robtarget Tr_meulage_motif_1_P265 :=[[-200.7086875,-41.05124609375,-0.0972945251464844],[0.732123189175605,-0.57971865199821,0.222030212103854,-0.280400615744397],[0,0,0,0],[8.999999E+09,8.999999E+09,8.999999E+09,8.999999E+09,8.999999E+09,8.999999E+09]];
	LOCAL CONST Robtarget Tr_meulage_motif_1_P266 :=[[-199.937109375,-41.68737890625,-0.0971960525512695],[0.732123189175605,-0.57971865199821,0.222030212103854,-0.280400615744397],[0,0,0,0],[8.999999E+09,8.999999E+09,8.999999E+09,8.999999E+09,8.999999E+09,8.999999E+09]];
	LOCAL CONST Robtarget Tr_meulage_motif_1_P267 :=[[-199.16553125,-42.32351171875,-0.0970975799560547],[0.732123189175605,-0.57971865199821,0.222030212103854,-0.280400615744397],[0,0,0,0],[8.999999E+09,8.999999E+09,8.999999E+09,8.999999E+09,8.999999E+09,8.999999E+09]];
	LOCAL CONST Robtarget Tr_meulage_motif_1_P268 :=[[-198.3939375,-42.95964453125,-0.0969991073608398],[0.732123189175605,-0.57971865199821,0.222030212103854,-0.280400615744397],[0,0,0,0],[8.999999E+09,8.999999E+09,8.999999E+09,8.999999E+09,8.999999E+09,8.999999E+09]];
	LOCAL CONST Robtarget Tr_meulage_motif_1_P269 :=[[-197.622359375,-43.59577734375,-0.096900634765625],[0.732123189175605,-0.57971865199821,0.222030212103854,-0.280400615744397],[0,0,0,0],[8.999999E+09,8.999999E+09,8.999999E+09,8.999999E+09,8.999999E+09,8.999999E+09]];
	LOCAL CONST Robtarget Tr_meulage_motif_1_P270 :=[[-196.85078125,-44.2319140625,-0.0968021621704102],[0.732123189175605,-0.57971865199821,0.222030212103854,-0.280400615744397],[0,0,0,0],[8.999999E+09,8.999999E+09,8.999999E+09,8.999999E+09,8.999999E+09,8.999999E+09]];
	LOCAL CONST Robtarget Tr_meulage_motif_1_P271 :=[[-196.079203125,-44.868046875,-0.0967036895751953],[0.732123189175605,-0.57971865199821,0.222030212103854,-0.280400615744397],[0,0,0,0],[8.999999E+09,8.999999E+09,8.999999E+09,8.999999E+09,8.999999E+09,8.999999E+09]];
	LOCAL CONST Robtarget Tr_meulage_motif_1_P272 :=[[-195.307625,-45.5041796875,-0.0966052169799805],[0.732123189175605,-0.57971865199821,0.222030212103854,-0.280400615744397],[0,0,0,0],[8.999999E+09,8.999999E+09,8.999999E+09,8.999999E+09,8.999999E+09,8.999999E+09]];
	LOCAL CONST Robtarget Tr_meulage_motif_1_P273 :=[[-194.536046875,-46.1403125,-0.0965067443847656],[0.732123189175605,-0.57971865199821,0.222030212103854,-0.280400615744397],[0,0,0,0],[8.999999E+09,8.999999E+09,8.999999E+09,8.999999E+09,8.999999E+09,8.999999E+09]];
	LOCAL CONST Robtarget Tr_meulage_motif_1_P274 :=[[-193.76446875,-46.7764453125,-0.0964082717895508],[0.732123189175605,-0.57971865199821,0.222030212103854,-0.280400615744397],[0,0,0,0],[8.999999E+09,8.999999E+09,8.999999E+09,8.999999E+09,8.999999E+09,8.999999E+09]];
	LOCAL CONST Robtarget Tr_meulage_motif_1_P275 :=[[-192.992890625,-47.412578125,-0.0963097991943359],[0.732123189175605,-0.57971865199821,0.222030212103854,-0.280400615744397],[0,0,0,0],[8.999999E+09,8.999999E+09,8.999999E+09,8.999999E+09,8.999999E+09,8.999999E+09]];
	LOCAL CONST Robtarget Tr_meulage_motif_1_P276 :=[[-192.2213125,-48.0487109375,-0.0962113265991211],[0.732123189175605,-0.57971865199821,0.222030212103854,-0.280400615744397],[0,0,0,0],[8.999999E+09,8.999999E+09,8.999999E+09,8.999999E+09,8.999999E+09,8.999999E+09]];
	LOCAL CONST Robtarget Tr_meulage_motif_1_P277 :=[[-191.449734375,-48.68484375,-0.0961128540039062],[0.732123189175605,-0.57971865199821,0.222030212103854,-0.280400615744397],[0,0,0,0],[8.999999E+09,8.999999E+09,8.999999E+09,8.999999E+09,8.999999E+09,8.999999E+09]];
	LOCAL CONST Robtarget Tr_meulage_motif_1_P278 :=[[-190.67815625,-49.3209765625,-0.0960143814086914],[0.732123189175605,-0.57971865199821,0.222030212103854,-0.280400615744397],[0,0,0,0],[8.999999E+09,8.999999E+09,8.999999E+09,8.999999E+09,8.999999E+09,8.999999E+09]];
	LOCAL CONST Robtarget Tr_meulage_motif_1_P279 :=[[-189.906578125,-49.95711328125,-0.0959159088134766],[0.732123189175605,-0.57971865199821,0.222030212103854,-0.280400615744397],[0,0,0,0],[8.999999E+09,8.999999E+09,8.999999E+09,8.999999E+09,8.999999E+09,8.999999E+09]];
	LOCAL CONST Robtarget Tr_meulage_motif_1_P280 :=[[-189.135,-50.59324609375,-0.0958174362182617],[0.732123189175605,-0.57971865199821,0.222030212103854,-0.280400615744397],[0,0,0,0],[8.999999E+09,8.999999E+09,8.999999E+09,8.999999E+09,8.999999E+09,8.999999E+09]];
	LOCAL CONST Robtarget Tr_meulage_motif_1_P281 :=[[-188.363421875,-51.22937890625,-0.0957189636230469],[0.732123189175605,-0.57971865199821,0.222030212103854,-0.280400615744397],[0,0,0,0],[8.999999E+09,8.999999E+09,8.999999E+09,8.999999E+09,8.999999E+09,8.999999E+09]];
	LOCAL CONST Robtarget Tr_meulage_motif_1_P282 :=[[-187.591828125,-51.86551171875,-0.095620491027832],[0.732123189175605,-0.57971865199821,0.222030212103854,-0.280400615744397],[0,0,0,0],[8.999999E+09,8.999999E+09,8.999999E+09,8.999999E+09,8.999999E+09,8.999999E+09]];
	LOCAL CONST Robtarget Tr_meulage_motif_1_P283 :=[[-186.82025,-52.50164453125,-0.0955220184326172],[0.732123189175605,-0.57971865199821,0.222030212103854,-0.280400615744397],[0,0,0,0],[8.999999E+09,8.999999E+09,8.999999E+09,8.999999E+09,8.999999E+09,8.999999E+09]];
	LOCAL CONST Robtarget Tr_meulage_motif_1_P284 :=[[-186.048671875,-53.13777734375,-0.0954235458374023],[0.732123189175605,-0.57971865199821,0.222030212103854,-0.280400615744397],[0,0,0,0],[8.999999E+09,8.999999E+09,8.999999E+09,8.999999E+09,8.999999E+09,8.999999E+09]];
	LOCAL CONST Robtarget Tr_meulage_motif_1_P285 :=[[-185.27709375,-53.77391015625,-0.0953250732421875],[0.732123189175605,-0.57971865199821,0.222030212103854,-0.280400615744397],[0,0,0,0],[8.999999E+09,8.999999E+09,8.999999E+09,8.999999E+09,8.999999E+09,8.999999E+09]];
	LOCAL CONST Robtarget Tr_meulage_motif_1_P286 :=[[-184.505515625,-54.41004296875,-0.0952266082763672],[0.732123189175605,-0.57971865199821,0.222030212103854,-0.280400615744397],[0,0,0,0],[8.999999E+09,8.999999E+09,8.999999E+09,8.999999E+09,8.999999E+09,8.999999E+09]];
	LOCAL CONST Robtarget Tr_meulage_motif_1_P287 :=[[-183.7339375,-55.04617578125,-0.0951281356811523],[0.732123189175605,-0.57971865199821,0.222030212103854,-0.280400615744397],[0,0,0,0],[8.999999E+09,8.999999E+09,8.999999E+09,8.999999E+09,8.999999E+09,8.999999E+09]];
	LOCAL CONST Robtarget Tr_meulage_motif_1_P288 :=[[-182.962359375,-55.68230859375,-0.0950296630859375],[0.732123189175605,-0.57971865199821,0.222030212103854,-0.280400615744397],[0,0,0,0],[8.999999E+09,8.999999E+09,8.999999E+09,8.999999E+09,8.999999E+09,8.999999E+09]];
	LOCAL CONST Robtarget Tr_meulage_motif_1_P289 :=[[-182.19078125,-56.3184453125,-0.0949311904907227],[0.732123189175605,-0.57971865199821,0.222030212103854,-0.280400615744397],[0,0,0,0],[8.999999E+09,8.999999E+09,8.999999E+09,8.999999E+09,8.999999E+09,8.999999E+09]];
	LOCAL CONST Robtarget Tr_meulage_motif_1_P290 :=[[-181.419203125,-56.954578125,-0.0948327178955078],[0.732123189175605,-0.57971865199821,0.222030212103854,-0.280400615744397],[0,0,0,0],[8.999999E+09,8.999999E+09,8.999999E+09,8.999999E+09,8.999999E+09,8.999999E+09]];
	LOCAL CONST Robtarget Tr_meulage_motif_1_P291 :=[[-180.647625,-57.5907109375,-0.094734245300293],[0.732123189175605,-0.57971865199821,0.222030212103854,-0.280400615744397],[0,0,0,0],[8.999999E+09,8.999999E+09,8.999999E+09,8.999999E+09,8.999999E+09,8.999999E+09]];
	LOCAL CONST Robtarget Tr_meulage_motif_1_P292 :=[[-179.876046875,-58.22684375,-0.0946357727050781],[0.732123189175605,-0.57971865199821,0.222030212103854,-0.280400615744397],[0,0,0,0],[8.999999E+09,8.999999E+09,8.999999E+09,8.999999E+09,8.999999E+09,8.999999E+09]];
	LOCAL CONST Robtarget Tr_meulage_motif_1_P293 :=[[-179.10446875,-58.8629765625,-0.0945373001098633],[0.732123189175605,-0.57971865199821,0.222030212103854,-0.280400615744397],[0,0,0,0],[8.999999E+09,8.999999E+09,8.999999E+09,8.999999E+09,8.999999E+09,8.999999E+09]];
	LOCAL CONST Robtarget Tr_meulage_motif_1_P294 :=[[-178.332890625,-59.499109375,-0.0944388275146484],[0.732123189175605,-0.57971865199821,0.222030212103854,-0.280400615744397],[0,0,0,0],[8.999999E+09,8.999999E+09,8.999999E+09,8.999999E+09,8.999999E+09,8.999999E+09]];
	LOCAL CONST Robtarget Tr_meulage_motif_1_P295 :=[[-177.5613125,-60.1352421875,-0.0943403549194336],[0.732123189175605,-0.57971865199821,0.222030212103854,-0.280400615744397],[0,0,0,0],[8.999999E+09,8.999999E+09,8.999999E+09,8.999999E+09,8.999999E+09,8.999999E+09]];
	LOCAL CONST Robtarget Tr_meulage_motif_1_P296 :=[[-176.78971875,-60.771375,-0.0942418823242187],[0.732123189175605,-0.57971865199821,0.222030212103854,-0.280400615744397],[0,0,0,0],[8.999999E+09,8.999999E+09,8.999999E+09,8.999999E+09,8.999999E+09,8.999999E+09]];
	LOCAL CONST Robtarget Tr_meulage_motif_1_P297 :=[[-176.02,-61.3980859375,-0.204585601806641],[0.732123189175605,-0.57971865199821,0.222030212103854,-0.280400615744397],[0,0,0,0],[8.999999E+09,8.999999E+09,8.999999E+09,8.999999E+09,8.999999E+09,8.999999E+09]];
	LOCAL CONST Robtarget Tr_meulage_motif_1_P298 :=[[-175.28228125,-61.99122265625,-0.415359283447266],[0.732123189175605,-0.57971865199821,0.222030212103854,-0.280400615744397],[0,0,0,0],[8.999999E+09,8.999999E+09,8.999999E+09,8.999999E+09,8.999999E+09,8.999999E+09]];
	LOCAL CONST Robtarget Tr_meulage_motif_1_P299 :=[[-174.614796875,-62.52212890625,-0.686690734863281],[0.732123189175605,-0.57971865199821,0.222030212103854,-0.280400615744397],[0,0,0,0],[8.999999E+09,8.999999E+09,8.999999E+09,8.999999E+09,8.999999E+09,8.999999E+09]];
	LOCAL CONST Robtarget Tr_meulage_motif_1_P300 :=[[-174.02646875,-62.98748046875,-0.962135498046875],[0.732123189175605,-0.57971865199821,0.222030212103854,-0.280400615744397],[0,0,0,0],[8.999999E+09,8.999999E+09,8.999999E+09,8.999999E+09,8.999999E+09,8.999999E+09]];
	LOCAL CONST Robtarget Tr_meulage_motif_1_P301 :=[[-173.15528125,-63.66175390625,-1.57721667480469],[0.732123189175605,-0.57971865199821,0.222030212103854,-0.280400615744397],[0,0,0,0],[8.999999E+09,8.999999E+09,8.999999E+09,8.999999E+09,8.999999E+09,8.999999E+09]];
	LOCAL CONST Robtarget Tr_meulage_motif_1_P302 :=[[-172.335515625,-64.27710546875,-2.4234697265625],[0.732123189175605,-0.57971865199821,0.222030212103854,-0.280400615744397],[0,0,0,0],[8.999999E+09,8.999999E+09,8.999999E+09,8.999999E+09,8.999999E+09,8.999999E+09]];
	LOCAL CONST Robtarget Tr_meulage_motif_1_P303 :=[[-171.64553125,-64.772875,-3.44569116210937],[0.732123189175605,-0.57971865199821,0.222030212103854,-0.280400615744397],[0,0,0,0],[8.999999E+09,8.999999E+09,8.999999E+09,8.999999E+09,8.999999E+09,8.999999E+09]];
	LOCAL CONST Robtarget Tr_meulage_motif_1_P304 :=[[-171.2296875,-65.0360390625,-4.5601826171875],[0.732123189175605,-0.57971865199821,0.222030212103854,-0.280400615744397],[0,0,0,0],[8.999999E+09,8.999999E+09,8.999999E+09,8.999999E+09,8.999999E+09,8.999999E+09]];
	LOCAL CONST Robtarget Tr_meulage_motif_1_P305 :=[[-171.184359375,-65.02371875,-5.25506103515625],[0.732123189175605,-0.57971865199821,0.222030212103854,-0.280400615744397],[0,0,0,0],[8.999999E+09,8.999999E+09,8.999999E+09,8.999999E+09,8.999999E+09,8.999999E+09]];
	LOCAL CONST Robtarget Tr_meulage_motif_1_P306 :=[[-171.161140625,-64.99565625,-5.91533837890625],[0.732123189175605,-0.57971865199821,0.222030212103854,-0.280400615744397],[0,0,0,0],[8.999999E+09,8.999999E+09,8.999999E+09,8.999999E+09,8.999999E+09,8.999999E+09]];
	LOCAL CONST Robtarget Tr_meulage_motif_1_P307 :=[[-171.180265625,-64.9326953125,-6.57541845703125],[0.732123189175605,-0.57971865199821,0.222030212103854,-0.280400615744397],[0,0,0,0],[8.999999E+09,8.999999E+09,8.999999E+09,8.999999E+09,8.999999E+09,8.999999E+09]];
	LOCAL CONST Robtarget Tr_meulage_motif_1_P308 :=[[-171.526,-64.5690078125,-7.675529296875],[0.732123189175605,-0.57971865199821,0.222030212103854,-0.280400615744397],[0,0,0,0],[8.999999E+09,8.999999E+09,8.999999E+09,8.999999E+09,8.999999E+09,8.999999E+09]];
	LOCAL CONST Robtarget Tr_meulage_motif_1_P309 :=[[-172.15159375,-63.981359375,-8.6807255859375],[0.732123189175605,-0.57971865199821,0.222030212103854,-0.280400615744397],[0,0,0,0],[8.999999E+09,8.999999E+09,8.999999E+09,8.999999E+09,8.999999E+09,8.999999E+09]];
	LOCAL CONST Robtarget Tr_meulage_motif_1_P310 :=[[-172.912140625,-63.2951640625,-9.508427734375],[0.732123189175605,-0.57971865199821,0.222030212103854,-0.280400615744397],[0,0,0,0],[8.999999E+09,8.999999E+09,8.999999E+09,8.999999E+09,8.999999E+09,8.999999E+09]];
	LOCAL CONST Robtarget Tr_meulage_motif_1_P311 :=[[-173.428390625,-62.84128515625,-9.90366015625],[0.732123189175605,-0.57971865199821,0.222030212103854,-0.280400615744397],[0,0,0,0],[8.999999E+09,8.999999E+09,8.999999E+09,8.999999E+09,8.999999E+09,8.999999E+09]];
	LOCAL CONST Robtarget Tr_meulage_motif_1_P312 :=[[-174.304875,-62.0838515625,-10.3905654296875],[0.732123189175605,-0.57971865199821,0.222030212103854,-0.280400615744397],[0,0,0,0],[8.999999E+09,8.999999E+09,8.999999E+09,8.999999E+09,8.999999E+09,8.999999E+09]];
	LOCAL CONST Robtarget Tr_meulage_motif_1_P313 :=[[-174.947609375,-61.53509375,-10.654357421875],[0.732123189175605,-0.57971865199821,0.222030212103854,-0.280400615744397],[0,0,0,0],[8.999999E+09,8.999999E+09,8.999999E+09,8.999999E+09,8.999999E+09,8.999999E+09]];
	LOCAL CONST Robtarget Tr_meulage_motif_1_P314 :=[[-175.659546875,-60.9335390625,-10.858623046875],[0.732123189175605,-0.57971865199821,0.222030212103854,-0.280400615744397],[0,0,0,0],[8.999999E+09,8.999999E+09,8.999999E+09,8.999999E+09,8.999999E+09,8.999999E+09]];
	LOCAL CONST Robtarget Tr_meulage_motif_1_P315 :=[[-176.413078125,-60.30452734375,-10.9671015625],[0.732123189175605,-0.57971865199821,0.222030212103854,-0.280400615744397],[0,0,0,0],[8.999999E+09,8.999999E+09,8.999999E+09,8.999999E+09,8.999999E+09,8.999999E+09]];
	LOCAL CONST Robtarget Tr_meulage_motif_1_P316 :=[[-177.17503125,-59.6684296875,-11.077640625],[0.732123189175605,-0.57971865199821,0.222030212103854,-0.280400615744397],[0,0,0,0],[8.999999E+09,8.999999E+09,8.999999E+09,8.999999E+09,8.999999E+09,8.999999E+09]];
	LOCAL CONST Robtarget Tr_meulage_motif_1_P317 :=[[-177.946609375,-59.032296875,-11.0777392578125],[0.732123189175605,-0.57971865199821,0.222030212103854,-0.280400615744397],[0,0,0,0],[8.999999E+09,8.999999E+09,8.999999E+09,8.999999E+09,8.999999E+09,8.999999E+09]];
	LOCAL CONST Robtarget Tr_meulage_motif_1_P318 :=[[-178.718203125,-58.3961640625,-11.077837890625],[0.732123189175605,-0.57971865199821,0.222030212103854,-0.280400615744397],[0,0,0,0],[8.999999E+09,8.999999E+09,8.999999E+09,8.999999E+09,8.999999E+09,8.999999E+09]];
	LOCAL CONST Robtarget Tr_meulage_motif_1_P319 :=[[-179.48978125,-57.76003125,-11.077935546875],[0.732123189175605,-0.57971865199821,0.222030212103854,-0.280400615744397],[0,0,0,0],[8.999999E+09,8.999999E+09,8.999999E+09,8.999999E+09,8.999999E+09,8.999999E+09]];
	LOCAL CONST Robtarget Tr_meulage_motif_1_P320 :=[[-180.261359375,-57.1238984375,-11.0780341796875],[0.732123189175605,-0.57971865199821,0.222030212103854,-0.280400615744397],[0,0,0,0],[8.999999E+09,8.999999E+09,8.999999E+09,8.999999E+09,8.999999E+09,8.999999E+09]];
	LOCAL CONST Robtarget Tr_meulage_motif_1_P321 :=[[-181.0329375,-56.487765625,-11.0781328125],[0.732123189175605,-0.57971865199821,0.222030212103854,-0.280400615744397],[0,0,0,0],[8.999999E+09,8.999999E+09,8.999999E+09,8.999999E+09,8.999999E+09,8.999999E+09]];
	LOCAL CONST Robtarget Tr_meulage_motif_1_P322 :=[[-181.804515625,-55.8516328125,-11.0782314453125],[0.732123189175605,-0.57971865199821,0.222030212103854,-0.280400615744397],[0,0,0,0],[8.999999E+09,8.999999E+09,8.999999E+09,8.999999E+09,8.999999E+09,8.999999E+09]];
	LOCAL CONST Robtarget Tr_meulage_motif_1_P323 :=[[-182.57609375,-55.2155,-11.078330078125],[0.732123189175605,-0.57971865199821,0.222030212103854,-0.280400615744397],[0,0,0,0],[8.999999E+09,8.999999E+09,8.999999E+09,8.999999E+09,8.999999E+09,8.999999E+09]];
	LOCAL CONST Robtarget Tr_meulage_motif_1_P324 :=[[-183.347671875,-54.5793671875,-11.0784287109375],[0.732123189175605,-0.57971865199821,0.222030212103854,-0.280400615744397],[0,0,0,0],[8.999999E+09,8.999999E+09,8.999999E+09,8.999999E+09,8.999999E+09,8.999999E+09]];
	LOCAL CONST Robtarget Tr_meulage_motif_1_P325 :=[[-184.11925,-53.943234375,-11.07852734375],[0.732123189175605,-0.57971865199821,0.222030212103854,-0.280400615744397],[0,0,0,0],[8.999999E+09,8.999999E+09,8.999999E+09,8.999999E+09,8.999999E+09,8.999999E+09]];
	LOCAL CONST Robtarget Tr_meulage_motif_1_P326 :=[[-184.890828125,-53.30709765625,-11.078625],[0.732123189175605,-0.57971865199821,0.222030212103854,-0.280400615744397],[0,0,0,0],[8.999999E+09,8.999999E+09,8.999999E+09,8.999999E+09,8.999999E+09,8.999999E+09]];
	LOCAL CONST Robtarget Tr_meulage_motif_1_P327 :=[[-185.66240625,-52.67096484375,-11.0787236328125],[0.732123189175605,-0.57971865199821,0.222030212103854,-0.280400615744397],[0,0,0,0],[8.999999E+09,8.999999E+09,8.999999E+09,8.999999E+09,8.999999E+09,8.999999E+09]];
	LOCAL CONST Robtarget Tr_meulage_motif_1_P328 :=[[-186.433984375,-52.03483203125,-11.078822265625],[0.732123189175605,-0.57971865199821,0.222030212103854,-0.280400615744397],[0,0,0,0],[8.999999E+09,8.999999E+09,8.999999E+09,8.999999E+09,8.999999E+09,8.999999E+09]];
	LOCAL CONST Robtarget Tr_meulage_motif_1_P329 :=[[-187.2055625,-51.39869921875,-11.0789208984375],[0.732123189175605,-0.57971865199821,0.222030212103854,-0.280400615744397],[0,0,0,0],[8.999999E+09,8.999999E+09,8.999999E+09,8.999999E+09,8.999999E+09,8.999999E+09]];
	LOCAL CONST Robtarget Tr_meulage_motif_1_P330 :=[[-187.977140625,-50.76256640625,-11.07901953125],[0.732123189175605,-0.57971865199821,0.222030212103854,-0.280400615744397],[0,0,0,0],[8.999999E+09,8.999999E+09,8.999999E+09,8.999999E+09,8.999999E+09,8.999999E+09]];
	LOCAL CONST Robtarget Tr_meulage_motif_1_P331 :=[[-188.74871875,-50.12643359375,-11.0791181640625],[0.732123189175605,-0.57971865199821,0.222030212103854,-0.280400615744397],[0,0,0,0],[8.999999E+09,8.999999E+09,8.999999E+09,8.999999E+09,8.999999E+09,8.999999E+09]];
	LOCAL CONST Robtarget Tr_meulage_motif_1_P332 :=[[-189.5203125,-49.49030078125,-11.0792158203125],[0.732123189175605,-0.57971865199821,0.222030212103854,-0.280400615744397],[0,0,0,0],[8.999999E+09,8.999999E+09,8.999999E+09,8.999999E+09,8.999999E+09,8.999999E+09]];
	LOCAL CONST Robtarget Tr_meulage_motif_1_P333 :=[[-190.291890625,-48.85416796875,-11.079314453125],[0.732123189175605,-0.57971865199821,0.222030212103854,-0.280400615744397],[0,0,0,0],[8.999999E+09,8.999999E+09,8.999999E+09,8.999999E+09,8.999999E+09,8.999999E+09]];
	LOCAL CONST Robtarget Tr_meulage_motif_1_P334 :=[[-191.06346875,-48.21803515625,-11.0794130859375],[0.732123189175605,-0.57971865199821,0.222030212103854,-0.280400615744397],[0,0,0,0],[8.999999E+09,8.999999E+09,8.999999E+09,8.999999E+09,8.999999E+09,8.999999E+09]];
	LOCAL CONST Robtarget Tr_meulage_motif_1_P335 :=[[-191.835046875,-47.5818984375,-11.07951171875],[0.732123189175605,-0.57971865199821,0.222030212103854,-0.280400615744397],[0,0,0,0],[8.999999E+09,8.999999E+09,8.999999E+09,8.999999E+09,8.999999E+09,8.999999E+09]];
	LOCAL CONST Robtarget Tr_meulage_motif_1_P336 :=[[-192.606625,-46.945765625,-11.0796103515625],[0.732123189175605,-0.57971865199821,0.222030212103854,-0.280400615744397],[0,0,0,0],[8.999999E+09,8.999999E+09,8.999999E+09,8.999999E+09,8.999999E+09,8.999999E+09]];
	LOCAL CONST Robtarget Tr_meulage_motif_1_P337 :=[[-193.378203125,-46.3096328125,-11.079708984375],[0.732123189175605,-0.57971865199821,0.222030212103854,-0.280400615744397],[0,0,0,0],[8.999999E+09,8.999999E+09,8.999999E+09,8.999999E+09,8.999999E+09,8.999999E+09]];
	LOCAL CONST Robtarget Tr_meulage_motif_1_P338 :=[[-194.14978125,-45.6735,-11.079806640625],[0.732123189175605,-0.57971865199821,0.222030212103854,-0.280400615744397],[0,0,0,0],[8.999999E+09,8.999999E+09,8.999999E+09,8.999999E+09,8.999999E+09,8.999999E+09]];
	LOCAL CONST Robtarget Tr_meulage_motif_1_P339 :=[[-194.921359375,-45.0373671875,-11.0799052734375],[0.732123189175605,-0.57971865199821,0.222030212103854,-0.280400615744397],[0,0,0,0],[8.999999E+09,8.999999E+09,8.999999E+09,8.999999E+09,8.999999E+09,8.999999E+09]];
	LOCAL CONST Robtarget Tr_meulage_motif_1_P340 :=[[-195.6929375,-44.401234375,-11.08000390625],[0.732123189175605,-0.57971865199821,0.222030212103854,-0.280400615744397],[0,0,0,0],[8.999999E+09,8.999999E+09,8.999999E+09,8.999999E+09,8.999999E+09,8.999999E+09]];
	LOCAL CONST Robtarget Tr_meulage_motif_1_P341 :=[[-196.464515625,-43.7651015625,-11.0801025390625],[0.732123189175605,-0.57971865199821,0.222030212103854,-0.280400615744397],[0,0,0,0],[8.999999E+09,8.999999E+09,8.999999E+09,8.999999E+09,8.999999E+09,8.999999E+09]];
	LOCAL CONST Robtarget Tr_meulage_motif_1_P342 :=[[-197.23609375,-43.12896875,-11.080201171875],[0.732123189175605,-0.57971865199821,0.222030212103854,-0.280400615744397],[0,0,0,0],[8.999999E+09,8.999999E+09,8.999999E+09,8.999999E+09,8.999999E+09,8.999999E+09]];
	LOCAL CONST Robtarget Tr_meulage_motif_1_P343 :=[[-198.007671875,-42.4928359375,-11.0802998046875],[0.732123189175605,-0.57971865199821,0.222030212103854,-0.280400615744397],[0,0,0,0],[8.999999E+09,8.999999E+09,8.999999E+09,8.999999E+09,8.999999E+09,8.999999E+09]];
	LOCAL CONST Robtarget Tr_meulage_motif_1_P344 :=[[-198.77925,-41.856703125,-11.0803974609375],[0.732123189175605,-0.57971865199821,0.222030212103854,-0.280400615744397],[0,0,0,0],[8.999999E+09,8.999999E+09,8.999999E+09,8.999999E+09,8.999999E+09,8.999999E+09]];
	LOCAL CONST Robtarget Tr_meulage_motif_1_P345 :=[[-199.550828125,-41.22056640625,-11.08049609375],[0.732123189175605,-0.57971865199821,0.222030212103854,-0.280400615744397],[0,0,0,0],[8.999999E+09,8.999999E+09,8.999999E+09,8.999999E+09,8.999999E+09,8.999999E+09]];
	LOCAL CONST Robtarget Tr_meulage_motif_1_P346 :=[[-200.322421875,-40.58443359375,-11.0805947265625],[0.732123189175605,-0.57971865199821,0.222030212103854,-0.280400615744397],[0,0,0,0],[8.999999E+09,8.999999E+09,8.999999E+09,8.999999E+09,8.999999E+09,8.999999E+09]];
	LOCAL CONST Robtarget Tr_meulage_motif_1_P347 :=[[-201.094,-39.94830078125,-11.080693359375],[0.732123189175605,-0.57971865199821,0.222030212103854,-0.280400615744397],[0,0,0,0],[8.999999E+09,8.999999E+09,8.999999E+09,8.999999E+09,8.999999E+09,8.999999E+09]];
	LOCAL CONST Robtarget Tr_meulage_motif_1_P348 :=[[-201.865578125,-39.31216796875,-11.0807919921875],[0.732123189175605,-0.57971865199821,0.222030212103854,-0.280400615744397],[0,0,0,0],[8.999999E+09,8.999999E+09,8.999999E+09,8.999999E+09,8.999999E+09,8.999999E+09]];
	LOCAL CONST Robtarget Tr_meulage_motif_1_P349 :=[[-202.63715625,-38.67603515625,-11.080890625],[0.732123189175605,-0.57971865199821,0.222030212103854,-0.280400615744397],[0,0,0,0],[8.999999E+09,8.999999E+09,8.999999E+09,8.999999E+09,8.999999E+09,8.999999E+09]];
	LOCAL CONST Robtarget Tr_meulage_motif_1_P350 :=[[-203.408734375,-38.03990234375,-11.08098828125],[0.732123189175605,-0.57971865199821,0.222030212103854,-0.280400615744397],[0,0,0,0],[8.999999E+09,8.999999E+09,8.999999E+09,8.999999E+09,8.999999E+09,8.999999E+09]];
	LOCAL CONST Robtarget Tr_meulage_motif_1_P351 :=[[-204.1803125,-37.40376953125,-11.0810869140625],[0.732123189175605,-0.57971865199821,0.222030212103854,-0.280400615744397],[0,0,0,0],[8.999999E+09,8.999999E+09,8.999999E+09,8.999999E+09,8.999999E+09,8.999999E+09]];
	LOCAL CONST Robtarget Tr_meulage_motif_1_P352 :=[[-204.951890625,-36.76763671875,-11.081185546875],[0.732123189175605,-0.57971865199821,0.222030212103854,-0.280400615744397],[0,0,0,0],[8.999999E+09,8.999999E+09,8.999999E+09,8.999999E+09,8.999999E+09,8.999999E+09]];
	LOCAL CONST Robtarget Tr_meulage_motif_1_P353 :=[[-205.72346875,-36.13150390625,-11.0812841796875],[0.732123189175605,-0.57971865199821,0.222030212103854,-0.280400615744397],[0,0,0,0],[8.999999E+09,8.999999E+09,8.999999E+09,8.999999E+09,8.999999E+09,8.999999E+09]];
	LOCAL CONST Robtarget Tr_meulage_motif_1_P354 :=[[-206.495046875,-35.4953671875,-11.0813828125],[0.732123189175605,-0.57971865199821,0.222030212103854,-0.280400615744397],[0,0,0,0],[8.999999E+09,8.999999E+09,8.999999E+09,8.999999E+09,8.999999E+09,8.999999E+09]];
	LOCAL CONST Robtarget Tr_meulage_motif_1_P355 :=[[-207.266625,-34.859234375,-11.0814814453125],[0.732123189175605,-0.57971865199821,0.222030212103854,-0.280400615744397],[0,0,0,0],[8.999999E+09,8.999999E+09,8.999999E+09,8.999999E+09,8.999999E+09,8.999999E+09]];
	LOCAL CONST Robtarget Tr_meulage_motif_1_P356 :=[[-208.038203125,-34.2231015625,-11.0815791015625],[0.732123189175605,-0.57971865199821,0.222030212103854,-0.280400615744397],[0,0,0,0],[8.999999E+09,8.999999E+09,8.999999E+09,8.999999E+09,8.999999E+09,8.999999E+09]];
	LOCAL CONST Robtarget Tr_meulage_motif_1_P357 :=[[-208.80978125,-33.58696875,-11.081677734375],[0.732123189175605,-0.57971865199821,0.222030212103854,-0.280400615744397],[0,0,0,0],[8.999999E+09,8.999999E+09,8.999999E+09,8.999999E+09,8.999999E+09,8.999999E+09]];
	LOCAL CONST Robtarget Tr_meulage_motif_1_P358 :=[[-209.581359375,-32.9508359375,-11.0817763671875],[0.732123189175605,-0.57971865199821,0.222030212103854,-0.280400615744397],[0,0,0,0],[8.999999E+09,8.999999E+09,8.999999E+09,8.999999E+09,8.999999E+09,8.999999E+09]];
	LOCAL CONST Robtarget Tr_meulage_motif_1_P359 :=[[-210.343328125,-32.314740234375,-11.1923154296875],[0.732123189175605,-0.57971865199821,0.222030212103854,-0.280400615744397],[0,0,0,0],[8.999999E+09,8.999999E+09,8.999999E+09,8.999999E+09,8.999999E+09,8.999999E+09]];
	LOCAL CONST Robtarget Tr_meulage_motif_1_P360 :=[[-211.066203125,-31.703677734375,-11.403275390625],[0.732123189175605,-0.57971865199821,0.222030212103854,-0.280400615744397],[0,0,0,0],[8.999999E+09,8.999999E+09,8.999999E+09,8.999999E+09,8.999999E+09,8.999999E+09]];
	LOCAL CONST Robtarget Tr_meulage_motif_1_P361 :=[[-211.71459375,-31.14969921875,-11.674775390625],[0.732123189175605,-0.57971865199821,0.222030212103854,-0.280400615744397],[0,0,0,0],[8.999999E+09,8.999999E+09,8.999999E+09,8.999999E+09,8.999999E+09,8.999999E+09]];
	LOCAL CONST Robtarget Tr_meulage_motif_1_P362 :=[[-212.25290625,-30.68418359375,-11.9785244140625],[0.732123189175605,-0.57971865199821,0.222030212103854,-0.280400615744397],[0,0,0,0],[8.999999E+09,8.999999E+09,8.999999E+09,8.999999E+09,8.999999E+09,8.999999E+09]];
	LOCAL CONST Robtarget Tr_meulage_motif_1_P363 :=[[-213.0278125,-29.9980078125,-12.6401513671875],[0.732123189175605,-0.57971865199821,0.222030212103854,-0.280400615744397],[0,0,0,0],[8.999999E+09,8.999999E+09,8.999999E+09,8.999999E+09,8.999999E+09,8.999999E+09]];
	LOCAL CONST Robtarget Tr_meulage_motif_1_P364 :=[[-213.622,-29.441029296875,-13.5785859375],[0.732123189175605,-0.57971865199821,0.222030212103854,-0.280400615744397],[0,0,0,0],[8.999999E+09,8.999999E+09,8.999999E+09,8.999999E+09,8.999999E+09,8.999999E+09]];
	LOCAL CONST Robtarget Tr_meulage_motif_1_P365 :=[[-213.93359375,-29.109662109375,-14.620265625],[0.732123189175605,-0.57971865199821,0.222030212103854,-0.280400615744397],[0,0,0,0],[8.999999E+09,8.999999E+09,8.999999E+09,8.999999E+09,8.999999E+09,8.999999E+09]];
	LOCAL CONST Robtarget Tr_meulage_motif_1_P366 :=[[-213.82571875,-29.159875,-15.1619462890625],[0.732123189175605,-0.57971865199821,0.222030212103854,-0.280400615744397],[0,0,0,0],[8.999999E+09,8.999999E+09,8.999999E+09,8.999999E+09,8.999999E+09,8.999999E+09]];
	LOCAL CONST Robtarget Tr_meulage_motif_1_P367 :=[[-213.7649375,-29.187443359375,-15.4772880859375],[0.732123189175605,-0.57971865199821,0.222030212103854,-0.280400615744397],[0,0,0,0],[8.999999E+09,8.999999E+09,8.999999E+09,8.999999E+09,8.999999E+09,8.999999E+09]];
	LOCAL CONST Robtarget Tr_meulage_motif_1_P368 :=[[-213.42734375,-29.40719140625,-16.2965966796875],[0.732123189175605,-0.57971865199821,0.222030212103854,-0.280400615744397],[0,0,0,0],[8.999999E+09,8.999999E+09,8.999999E+09,8.999999E+09,8.999999E+09,8.999999E+09]];
	LOCAL CONST Robtarget Tr_meulage_motif_1_P369 :=[[-213.0964375,-29.6466484375,-16.76306640625],[0.732123189175605,-0.57971865199821,0.222030212103854,-0.280400615744397],[0,0,0,0],[8.999999E+09,8.999999E+09,8.999999E+09,8.999999E+09,8.999999E+09,8.999999E+09]];
	LOCAL CONST Robtarget Tr_meulage_motif_1_P370 :=[[-212.240125,-30.310421875,-17.35346875],[0.732123189175605,-0.57971865199821,0.222030212103854,-0.280400615744397],[0,0,0,0],[8.999999E+09,8.999999E+09,8.999999E+09,8.999999E+09,8.999999E+09,8.999999E+09]];
	LOCAL CONST Robtarget Tr_meulage_motif_1_P371 :=[[-211.592734375,-30.8230703125,-17.6484375],[0.732123189175605,-0.57971865199821,0.222030212103854,-0.280400615744397],[0,0,0,0],[8.999999E+09,8.999999E+09,8.999999E+09,8.999999E+09,8.999999E+09,8.999999E+09]];
	LOCAL CONST Robtarget Tr_meulage_motif_1_P372 :=[[-210.866453125,-31.407267578125,-17.85251953125],[0.732123189175605,-0.57971865199821,0.222030212103854,-0.280400615744397],[0,0,0,0],[8.999999E+09,8.999999E+09,8.999999E+09,8.999999E+09,8.999999E+09,8.999999E+09]];
